(* CODESYS project CtaAppVerdichter_2.0.0.0.library
   Description: Verdichter Library der CTA
   Version: 2.0.0.0
   Title: CtaAppVerdichter
   Author: SIS
   DocFormat: reStructuredText
   Placeholder: CtaAppVerdichter
   LanguageModelAttribute: qualified-access-only
   CompiledLibraryCompatibilityVersion: CODESYS V3.5 SP16 Patch 3
   Company: CTA
   DefaultNamespace: CtaAppVerdichter

Project tree, tasks and I/O mapping:
  libraries: Standard, 3.5.18.0 (System); CtaAppBasic, 1.0.0.0 (CTA); CtaAppBmk, 2.0.0.0 (CTA); CtaAppReport, 2.0.0.0 (CTA); CtaSysConfig, 2.0.0.0 (CTA); CtaVisSymbols, 2.0.0.0 (CTA); CtaAppFilter, 1.0.0.0 (CTA); CtaAppHysterese, 1.0.0.0 (CTA); CtaSysMotor, 1.0.0.0 (CTA); CtaSysFU, 2.0.0.0 (CTA); VisuElemBase, 4.7.0.0 (System); CtaVisHelp, 2.0.0.0 (CTA); CtaAppDumper, 2.0.0.0 (CTA); CtaSysTypes, 1.0.0.0 (CTA); VisuDialogs, * (System); CtaAppEinsatzDiagramm, 2.0.0.0 (CTA); VisuSymbols, 4.5.0.0 (System); CtaSysLeistungventile, 2.0.0.0 (CTA); CtaAppInfluxLog, 1.0.0.1 (CTA); CtaSysIO, 2.0.0.0 (CTA); CtaAppModbusSpezifikation, 1.0.0.1 (CTA)
  40 Visualizations/
    ICON/
      VERDICHTER_RIGHT/
        VERDICHTER_RIGHT_BELOW/
          visualisation VIS_VERDICHTER_RIGHT_BELOW
          visualisation VIS_VERDICHTER_RigthBelowCheckIsEnabled
          visualisation VIS_VERDICHTER_RigthBelowCheckQuerry
        VERDICHTER_RIGHT_ABOVE/
          visualisation VIS_VERDICHTER_RigthAboveCheckQuerry
          visualisation VIS_VERDICHTER_RIGHT_ABOVE
          visualisation VIS_VERDICHTER_RigthAboveCheckIsEnabled
      VERDICHTER_BASE/
        visualisation CommandOn
        VALUE/
          visualisation ValueUpDwn
          visualisation ValueDwnUp
        ICON/
          visualisation Icon_Left
          visualisation Icon_Right
      VERDICHTER_LEFT/
        VERDICHTER_LEFT_BELOW/
          visualisation VIS_VERDICHTER_LEFT_BELOW
          visualisation VIS_VERDICHTER_LeftBelowCheckIsEnabled
          visualisation VIS_VERDICHTER_LeftBelowCheckQuerry
        VERDICHTER_LEFT_ABOVE/
          visualisation VIS_VERDICHTER_LEFT_ABOVE
          visualisation VIS_VERDICHTER_LeftAboveCheckIsEnabled
          visualisation VIS_VERDICHTER_LeftAboveCheckQuerry
    POPUP/
      visualisation POPUP_VERDICHTER
      PARAMETER/
        visualisation VIS_VERDICHTER_PARAMETER
        visualisation VIS_VERDICHTER_PARAMETER_LISTE
        VERDICHTER_ParameterBase/
          visualisation VIS_VERDICHTER_PARAMETER_BASE0
          visualisation VIS_VERDICHTER_PARAMETER_BASE
        VERDICHTER_Data/
          visualisation VIS_VERDICHTER_PARAMETER_DATA0
          visualisation VIS_VERDICHTER_PARAMETER_DATA
        VERDICHTER_Fuse/
          visualisation VIS_VERDICHTER_PARAMETER_FUSES0
          visualisation VIS_VERDICHTER_PARAMETER_FUSES
        VERDICHTER_IO/
          visualisation VIS_VERDICHTER_PARAMETER_IO0
          visualisation VIS_VERDICHTER_PARAMETER_IO1
          visualisation VIS_VERDICHTER_PARAMETER_IO
          visualisation VIS_VERDICHTER_PARAMETER_IO2
          visualisation VIS_VERDICHTER_PARAMETER_IO3
          visualisation VIS_VERDICHTER_PARAMETER_IO4
        VERDICHTER_InfluxDb/
          visualisation VIS_VERDICHTER_PARAMETER_TRENDLOG
          visualisation VIS_VERDICHTER_PARAMETER_TRENDLOG0
        visualisation VIS_ANTRIEB_POPUP_IO_ITF
      visualisation VIS_VERDICHTER_LISTE
      MANUAL/
        visualisation VIS_VERDICHTER_MANUAL
      OVERVIEW/
        visualisation VIS_VERDICHTER_OVERVIEW
        visualisation ResetVerdiTime
      BUS/
        visualisation VERDICHTER_BUS
        visualisation VERDICHTER_BUS_SW0_Detail
        visualisation VERDICHTER_BUS_CS
        visualisation VERDICHTER_BUS_SW1_Detail
        visualisation VERDICHTER_BUS_SW2_Detail
        visualisation VERDICHTER_BUS_SW3_Detail
      REPORTS/
        visualisation VIS_VERDICHTER_REPORTS
      IO/
        visualisation VIS_VERDICHTER_IO0
        visualisation VIS_VERDICHTER_IO
        visualisation VIS_VERDICHTER_IO1
  30 Program Organization Units/
    function block fbVerdichter [ST]: actConfig, proConfigError, proAtIconNr, P_scBase_fbtDelayOffToOn, P_scBase_fbtDelayOnToOn, P_scBase_fbrYMax, P_scBase_fbrYMin, P_scBase_fbxEnableFU, P_scBase_fbxEnable, P_scBase_fbxRegulatet, P_scData_fbudiOperatingHours, P_scData_fbudiOperationStarts, P_scFuse_fbxDoesAlarm, P_scFuse_fbxEnable, P_scFuse_fbxInputMb, P_scInfluxDb_fbxEnable, P_scIO_IsHand_fbxEnable, P_scIO_IsHand_fbxInputMb, P_scIO_IsNoError_fbxEnable, P_scIO_IsNoError_fbxInputMb, P_scIO_IsNoError_fbxDoesAlarm, P_scIO_IsNoError_fbtDelayStartSps, P_scIO_IsNoError_fbtDelayRun, P_scIO_IsNoError_fbiTypeOfAck, P_scIO_IsNoError_fbiMaxErrorRetryAllowed, P_scIO_IsOn_fbxInputMb, P_scIO_IsOn_fbxEnable, P_scIO_IsOn_fbtDelayStart, P_scIO_IsOn_fbxDoesAlarm, P_scIO_IsOn_fbtDelayRun, P_scIO_IsOn_fbiTypeOfAck, P_scIO_IsOn_fbiMaxErrorRetryAllowed, P_scIO_IsReady_fbxEnable, P_scIO_IsReady_fbxInputMb, P_scIO_IsValue_fbxInputMb, P_scIO_IsValue_fbxEnable, P_scIO_IsValue_fbxDoesAlarm, P_scIO_IsValue_fbtDelayStart, P_scIO_IsValue_fbtDelayRun, P_scIO_IsValue_fbiTypeOfAck, P_scIO_IsValue_fbiMaxErrorRetryAllowed, P_scIO_IsValue_fbrMaxDiff, P_scIO_RevisionSwitch_fbxEnable, P_scIO_RevisionSwitch_fbxInputMb, P_scManual_fbrManualOnY, P_scManual_fbuiManualState, P_scManual_fbxAlowManualOn, P_scVerdichterFuse_fbxDoesAlarm, P_scVerdichterFuse_fbxEnable, P_scVerdichterFuse_fbxInputMb, P_scFU_fbxReleaseMb, P_scFU_fbxSollWertMb, proRefToRonYDumper, actMbState, proModbusTest, proModbusStateWord, proIsError, proIsWarning, proIsRegulatet, proIsEnabled, actState, proMotorIsOn, proIsHandOnOrOff, proIsReady, proRestartLockAktive, proCommutingProtectionAktive, proRevisionSwitchOk, proCountedHours, proCountedStarts, proLeistung, proRestartLockTime, proCommutingProtectionTime, proIsOnY, proStateSymbol, proEnSymbol, proIsOn, proResetVerdiTime, proAuto, proHandOff, proHandOnY, proHardWareHandModulAktive, proHandOn, proGetDI_IsOn, metDI_IsOn, proNotShowDI_IsOn, proIsOn_ITF, metDI_RevisionSwitchOk, proNotShowDI_RevisionSwitchOk, proGetDI_RevisionSwitchOK, proRevisionSwitch_ITF, metDI_NoError, proNotShowDI_NoError, proGetDI_NoError, proNoError_ITF, proGetDI_FuseOK, metDI_ITF_FuseOK, proNotShowDI_FuseOk, proFuse_ITF, metDI_ITF_VerdichterHand, proNotShowDI_VerdichterHand, proGetDI_VerdichterHand, proHandModul_ITF, metDI_IsReady, proNotShowDI_Ready, proGetDI_IsReady, proReady_ITF, metDI_VerdichterFuseOk, proNotShowDI_VerdichterFuseOk, proGetDI_VerdichterFuseOk, proVerdichterFuse_ITF, metAI_ActualValue, proGetAI_ActualValue, proNotShowAI_ActualValue, proActualValue_ITF, proOnY_ITF, metAO_OnY, proDO_On, metDO_On, proOn_ITF, proOnY, proOn, actRestartAndCommutingLock, actPrioOfControll, actResetOnDisable, proOnHz, proEn, actTrendLog, actReport, proCountedError, proCountedInfo, proCountedWarning, proITF_REPORTMANAGER, proLockDown, proAvailable, proAcknowledge, proITF_EINSATZGRENZE, proITF_FU, actFU, proITF_LEISTUNGVENTILE, actLeistungsventile
    function fcGetBigerStringValue [ST]
    function fcCheckQuerryAndIconReturn [ST]
  00000000-0000-0000-0000-000000000000|D:\CoDeSys\LibrariesV3\trunk\Intern\CAA\CAA Template\3.4.0.0 draft\Placeholder.xml
  00000000-0000-0000-0000-000000000000|D:\CoDeSys\LibrariesV3\trunk\Intern\CAA\CAA Template\3.2.0.3 draft\Prefix.pdf
  00000000-0000-0000-0000-000000000000|D:\CoDeSys\LibrariesV3\trunk\Intern\CAA\CAA Template\3.5.2.0 draft\Placeholder.xml
  20 Structs/
    Verdichter/
      FU/
        data type scFU
      data type scParameter
      STATE/
        data type scInVerdichterHand
        data type scInVerichterActualValue
        data type scInVerdiRevisionSwitch
        data type scInVerdichterReady
        data type scInVerdichterNoError
        data type scInVerdichterOn
      BASE/
        data type scBase
      DATA/
        data type scData
      FUSE/
        data type scVerdichterFuse
        data type scFuse
      InfluxDb/
        data type scInfluxDb
      MANUAL/
        data type scManual
    Einsatzgrenze/
      data type scParameterEinsatzgrenze
      Paint/
        data type scLinePoint
        data type scDiagrammSizePaint
      Parameter/
        data type scSlopValue1
        data type scSlopValue2
        data type scSlopValue3
        data type scSlopValue4
        data type scSlopValue5
        data type scSlopValue6
        data type scDiagrammSize
        data type scErrorWarning
  50 Images/
  10 Documenation/
    global variables VersionHistory
    global variables readMe
  21 Interface/
    interface ITF_VERDICHTER: proModbusTest, proModbusStateWord, P_scFU_fbxReleaseMb, P_scFU_fbxSollWertMb, proConfigError, proAtIconNr, P_scBase_fbxEnable, P_scBase_fbxRegulatet, P_scBase_fbxEnableFU, P_scBase_fbrYMax, P_scBase_fbrYMin, P_scBase_fbtDelayOnToOn, P_scBase_fbtDelayOffToOn, P_scData_fbudiOperatingHours, P_scData_fbudiOperationStarts, P_scFuse_fbxDoesAlarm, P_scFuse_fbxEnable, P_scFuse_fbxInputMb, P_scInfluxDb_fbxEnable, P_scIO_RevisionSwitch_fbxEnable, P_scIO_RevisionSwitch_fbxInputMb, P_scIO_IsReady_fbxEnable, P_scIO_IsReady_fbxInputMb, P_scIO_IsHand_fbxEnable, P_scIO_IsHand_fbxInputMb, P_scIO_IsOn_fbxInputMb, P_scIO_IsOn_fbxEnable, P_scIO_IsOn_fbtDelayStart, P_scIO_IsOn_fbxDoesAlarm, P_scIO_IsOn_fbtDelayRun, P_scIO_IsOn_fbiTypeOfAck, P_scIO_IsOn_fbiMaxErrorRetryAllowed, P_scIO_IsNoError_fbxEnable, P_scIO_IsNoError_fbxInputMb, P_scIO_IsNoError_fbxDoesAlarm, P_scIO_IsNoError_fbtDelayStartSps, P_scIO_IsNoError_fbtDelayRun, P_scIO_IsNoError_fbiTypeOfAck, P_scIO_IsNoError_fbiMaxErrorRetryAllowed, P_scIO_IsValue_fbxInputMb, P_scIO_IsValue_fbxEnable, P_scIO_IsValue_fbxDoesAlarm, P_scIO_IsValue_fbtDelayStart, P_scIO_IsValue_fbtDelayRun, P_scIO_IsValue_fbiTypeOfAck, P_scIO_IsValue_fbiMaxErrorRetryAllowed, P_scIO_IsValue_fbrMaxDiff, P_scManual_fbrManualOnY, P_scManual_fbuiManualState, P_scManual_fbxAlowManualOn, P_scVerdichterFuse_fbxDoesAlarm, P_scVerdichterFuse_fbxEnable, P_scVerdichterFuse_fbxInputMb, proRefToRonYDumper, proCountedError, proCountedInfo, proITF_REPORTMANAGER, proCountedWarning, proCountedHours, proCountedStarts, proGetDI_VerdichterHand, proNotShowDI_VerdichterHand, proHandModul_ITF, proGetAI_ActualValue, proNotShowAI_ActualValue, proActualValue_ITF, proNotShowDI_NoError, proGetDI_NoError, proNoError_ITF, proNotShowDI_RevisionSwitchOk, proGetDI_RevisionSwitchOK, proRevisionSwitch_ITF, proNotShowDI_IsOn, proGetDI_IsOn, proIsOn_ITF, proNotShowDI_VerdichterFuseOk, proGetDI_VerdichterFuseOk, proVerdichterFuse_ITF, proNotShowDI_FuseOk, proGetDI_FuseOK, proFuse_ITF, proNotShowDI_Ready, proGetDI_IsReady, proReady_ITF, proOn_ITF, proOnY_ITF, proLeistung, proIsOn, proIsOnY, proEnSymbol, proStateSymbol, proIsRegulatet, proIsHandOnOrOff, proRestartLockTime, proOn, proCommutingProtectionTime, proCommutingProtectionAktive, proRestartLockAktive, proIsReady, proAuto, proHandOn, proIsError, proIsWarning, proEn, proOnY, proHardWareHandModulAktive, proIsEnabled, proMotorIsOn, proHandOff, proRevisionSwitchOk, proHandOnY, proOnHz, proResetVerdiTime, proLockDown, proAvailable, proAcknowledge, proITF_EINSATZGRENZE, proITF_FU, proITF_LEISTUNGVENTILE
  11 Library Parameter/
    global variables Parameter
  12 Konstanten/
    global variables GlobalKonstant
  60 Textlisten/
    text list GlobalTextList
    text list Error
    text list Info
    text list Warnung
  13 Globale Variablen/
  5ce3da45-db07-42e7-a21c-a00fff4ed8f6|C:\Users\sis\Downloads\dip-switch.svg
  5ce3da45-db07-42e7-a21c-a00fff4ed8f6|C:\Users\sis\Downloads\lightning-bolt-circle.svg
  5ce3da45-db07-42e7-a21c-a00fff4ed8f6|C:\Users\sis\Downloads\sine-wave.svg
  5ce3da45-db07-42e7-a21c-a00fff4ed8f6|C:\Users\sis\Downloads\eye.svg
  5ce3da45-db07-42e7-a21c-a00fff4ed8f6|C:\Users\sis\Downloads\lan.svg
*)

// 20 Structs/Verdichter/scParameter
{attribute 'pack_mode' := '1'} 
TYPE scParameter :
    STRUCT
        scBase              		:   scBase;
        scFuse              		:   scFuse;
        scVerdichterFuse        	:   scVerdichterFuse;
        scInVerdiRevisionSwitch		:   scInVerdiRevisionSwitch;
        scInVerdichterReady     	:   scInVerdichterReady;
 		scInVerdichterHand      	:   scInVerdichterHand;   
        scInVerdichterOn    		:   scInVerdichterOn;
        scInVerdichterNoError   	:   scInVerdichterNoError;
        scInVerdichterActualValue  	:   scInVerichterActualValue;
        scManual            		:   scManual;
        scData              		:   scData;
        scInfluxDb          		:   scInfluxDb;       
		scFU						:	scFU;
    END_STRUCT
END_TYPE

// 20 Structs/Verdichter/STATE/scInVerdichterHand
{attribute 'pack_mode' := '1'} 
TYPE scInVerdichterHand :
    STRUCT
        fbxEnable                   : CtaSysConfig.fbBOOL;    
        fbxInputMb                  : CtaSysConfig.fbBOOL; 
    END_STRUCT
END_TYPE

// 20 Structs/Verdichter/STATE/scInVerichterActualValue
{attribute 'pack_mode' := '1'} 
TYPE scInVerichterActualValue :
    STRUCT
        fbxEnable                    : CtaSysConfig.fbBOOL;
        fbxInputMb                   : CtaSysConfig.fbBOOL;   
        fbxDoesAlarm                 : CtaSysConfig.fbBOOL;  
        fbrMaxDiff                   : CtaSysConfig.fbREAL;
        fbtDelayStart                : CtaSysConfig.fbTIME;
        fbtDelayRun                  : CtaSysConfig.fbTIME;
		fbiTypeOfAck				 : CtaSysConfig.fbINT;
		fbiMaxErrorRetryAllowed		 : CtaSysConfig.fbINT;          
    END_STRUCT
END_TYPE

// 20 Structs/Verdichter/STATE/scInVerdiRevisionSwitch
{attribute 'pack_mode' := '1'} 
TYPE scInVerdiRevisionSwitch :
    STRUCT
        fbxEnable                   : CtaSysConfig.fbBOOL;
        fbxInputMb                  : CtaSysConfig.fbBOOL;           
    END_STRUCT
END_TYPE

// 20 Structs/Verdichter/STATE/scInVerdichterReady
{attribute 'pack_mode' := '1'} 
TYPE scInVerdichterReady :
    STRUCT
        fbxEnable                    : CtaSysConfig.fbBOOL;
        fbxInputMb                   : CtaSysConfig.fbBOOL;
		fbxDoesAlarm				 : CtaSysConfig.fbBOOL;
		fbtDelayStart				 : CtaSysConfig.fbTIME;
		fbtDelayRun					 : CtaSysConfig.fbTIME;
		fbiTypeOfAck				 : CtaSysConfig.fbINT;
		fbiMaxErrorRetryAllowed		 : CtaSysConfig.fbINT;          
    END_STRUCT
END_TYPE

// 20 Structs/Verdichter/STATE/scInVerdichterNoError
{attribute 'pack_mode' := '1'} 
TYPE scInVerdichterNoError :
    STRUCT
        fbxEnable                    : CtaSysConfig.fbBOOL;
        fbxInputMb                   : CtaSysConfig.fbBOOL;   
        fbxDoesAlarm                 : CtaSysConfig.fbBOOL;  
        fbtDelayStartSps             : CtaSysConfig.fbTIME;
        fbtDelayRun                  : CtaSysConfig.fbTIME; 
        fbiTypeOfAck                 : CtaSysConfig.fbINT; 
        fbiMaxErrorRetryAllowed      : CtaSysConfig.fbINT; 
    END_STRUCT
END_TYPE

// 20 Structs/Verdichter/STATE/scInVerdichterOn
{attribute 'pack_mode' := '1'} 
TYPE scInVerdichterOn :
    STRUCT
        fbxEnable                    : CtaSysConfig.fbBOOL;
        fbxInputMb                   : CtaSysConfig.fbBOOL;   
        fbxDoesAlarm                 : CtaSysConfig.fbBOOL;  
        fbtDelayStart                : CtaSysConfig.fbTIME;
        fbtDelayRun                  : CtaSysConfig.fbTIME; 
        fbiTypeOfAck                 : CtaSysConfig.fbINT;   
        fbiMaxErrorRetryAllowed      : CtaSysConfig.fbINT;      
    END_STRUCT
END_TYPE

// 20 Structs/Verdichter/BASE/scBase
{attribute 'pack_mode' := '1'} 
TYPE scBase :
    STRUCT
        fbxEnable       :   CtaSysConfig.fbBOOL;
        fbxRegulatet    :   CtaSysConfig.fbBOOL;
        fbxEnableFU   	:   CtaSysConfig.fbBOOL;
        fbrYMin         :   CtaSysConfig.fbREAL;
        fbrYMax         :   CtaSysConfig.fbREAL;
        fbtDelayOffToOn :   CtaSysConfig.fbTIME;
        fbtDelayOnToOn 	:   CtaSysConfig.fbTIME;
    END_STRUCT
END_TYPE

// 20 Structs/Verdichter/DATA/scData
{attribute 'pack_mode' := '1'} 
TYPE scData :
    STRUCT
        fbudiOperationStarts    :   CtaSysConfig.fbUDINT;
        fbudiOperatingHours     :   CtaSysConfig.fbUDINT;       
    END_STRUCT
END_TYPE

// 20 Structs/Verdichter/FUSE/scVerdichterFuse
{attribute 'pack_mode' := '1'} 
TYPE scVerdichterFuse :
    STRUCT
        fbxEnable             : CtaSysConfig.fbBOOL;
        fbxInputMb            : CtaSysConfig.fbBOOL;
        fbxDoesAlarm          : CtaSysConfig.fbBOOL;      
    END_STRUCT
END_TYPE

// 20 Structs/Verdichter/FUSE/scFuse
{attribute 'pack_mode' := '1'} 
TYPE scFuse :
    STRUCT
        fbxEnable               : CtaSysConfig.fbBOOL;
        fbxInputMb              : CtaSysConfig.fbBOOL;
        fbxDoesAlarm            : CtaSysConfig.fbBOOL;
    END_STRUCT
END_TYPE

// 20 Structs/Verdichter/InfluxDb/scInfluxDb
{attribute 'pack_mode' := '1'} 
TYPE scInfluxDb :
    STRUCT
        fbxEnable       :   CtaSysConfig.fbBOOL;
    END_STRUCT
END_TYPE

// 20 Structs/Verdichter/MANUAL/scManual
{attribute 'pack_mode' := '1'} 
TYPE scManual :
    STRUCT
        fbxAlowManualOn         : CtaSysConfig.fbBOOL;    
        fbuiManualState         : CtaSysConfig.fbUINT;            // 0 = Auto ; 1 = Manual Off 2 = Manual On
        fbrManualOnY            : CtaSysConfig.fbREAL; 
    END_STRUCT
END_TYPE

// 20 Structs/Verdichter/FU/scFU
TYPE scFU :
	STRUCT
		fbxReleaseMb            : CtaSysConfig.fbBOOL;
		fbxSollWertMb           : CtaSysConfig.fbBOOL;
	END_STRUCT
END_TYPE

// 20 Structs/Einsatzgrenze/scParameterEinsatzgrenze
TYPE scParameterEinsatzgrenze :
    STRUCT
        scDiagrammSize              :   scDiagrammSize;
        fbrMinTc					:	CtaSysConfig.fbREAL;							        // Minimale Kondensationstemperatur [°C] 
        fbrMaxTc					:	CtaSysConfig.fbREAL;							        // Maximale Kondensationstemperatur [°C] 
        fbrMinTo					:	CtaSysConfig.fbREAL;							        // Minimale Verdampfungstemperatur  [°C]
        fbrMaxTo					:	CtaSysConfig.fbREAL; 							        // Maximale Verdampfungstemperatur  [°C]             
        scSlopValue1                :   scSlopValue1;         
        scSlopValue2                :   scSlopValue2;
        scSlopValue3                :   scSlopValue3;
        scSlopValue4                :   scSlopValue4;
        scSlopValue5                :   scSlopValue5;
        scSlopValue6                :   scSlopValue6;        
        scErrorWarning              :   scErrorWarning; 
    END_STRUCT
END_TYPE

// 20 Structs/Einsatzgrenze/Paint/scLinePoint
TYPE scLinePoint :
    STRUCT
        rP1X        :   REAL;
        rP1Y        :   REAL;      
    END_STRUCT
END_TYPE

// 20 Structs/Einsatzgrenze/Paint/scDiagrammSizePaint
TYPE scDiagrammSizePaint :
    STRUCT
        rYMax   :   REAL;
        rYMin   :   REAL;
        rXMax   :   REAL;
        rXMin   :   REAL;    
    END_STRUCT
END_TYPE

// 20 Structs/Einsatzgrenze/Parameter/scSlopValue1
TYPE scSlopValue1 :
    STRUCT
        fbrTcL			    :	CtaSysConfig.fbREAL;							        // Punkt  1 Kompressor-Auslegungsdiagramm [°C] 
        fbrT0L              :   CtaSysConfig.fbREAL;	                                // Punkt  2 Kompressor-Auslegungsdiagramm [°C]
        fbrT0R  		    :	CtaSysConfig.fbREAL;							        // Punkt  3 Kompressor-Auslegungsdiagramm [°C]        
    END_STRUCT
END_TYPE

// 20 Structs/Einsatzgrenze/Parameter/scSlopValue2
TYPE scSlopValue2 :
    STRUCT
        fbrTcR			    :	CtaSysConfig.fbREAL;							        // Punkt  4 Kompressor-Auslegungsdiagramm [°C] 
        fbrT0R  		    :	CtaSysConfig.fbREAL;							        // Punkt  5 Kompressor-Auslegungsdiagramm [°C]        
    END_STRUCT
END_TYPE

// 20 Structs/Einsatzgrenze/Parameter/scSlopValue3
TYPE scSlopValue3 :
    STRUCT
        fbrTcU			    :	CtaSysConfig.fbREAL;							        // Punkt  6 Kompressor-Auslegungsdiagramm [°C] 
    END_STRUCT
END_TYPE

// 20 Structs/Einsatzgrenze/Parameter/scSlopValue4
TYPE scSlopValue4 :
    STRUCT
        fbrTcL			    :	CtaSysConfig.fbREAL;							        // Punkt  7 Kompressor-Auslegungsdiagramm [°C]         
    END_STRUCT
END_TYPE

// 20 Structs/Einsatzgrenze/Parameter/scSlopValue5
TYPE scSlopValue5 :
    STRUCT
        fbrT0L			    :	CtaSysConfig.fbREAL;							        // Punkt  8 Kompressor-Auslegungsdiagramm [°C] 
        fbrT0R  			:	CtaSysConfig.fbREAL;							        // Punkt  9 Kompressor-Auslegungsdiagramm [°C]                
    END_STRUCT
END_TYPE

// 20 Structs/Einsatzgrenze/Parameter/scSlopValue6
TYPE scSlopValue6 :
    STRUCT
        fbrTcO			    :	CtaSysConfig.fbREAL;							        // Punkt 10 Kompressor-Auslegungsdiagramm [°C]                 
    END_STRUCT
END_TYPE

// 20 Structs/Einsatzgrenze/Parameter/scDiagrammSize
TYPE scDiagrammSize :
    STRUCT
        fbrYMax   :   CtaSysConfig.fbREAL;
        fbrYMin   :   CtaSysConfig.fbREAL;
        fbrXMax   :   CtaSysConfig.fbREAL;
        fbrXMin   :   CtaSysConfig.fbREAL;    
    END_STRUCT
END_TYPE

// 20 Structs/Einsatzgrenze/Parameter/scErrorWarning
TYPE scErrorWarning :
    STRUCT
        fbxEnEW1          :   CtaSysConfig.fbBOOL;
        fbxEnEW2          :   CtaSysConfig.fbBOOL;
        fbxEnEW3          :   CtaSysConfig.fbBOOL;
        fbxEnEW4          :   CtaSysConfig.fbBOOL;
        fbxEnEW5          :   CtaSysConfig.fbBOOL;
        fbxEnEW6          :   CtaSysConfig.fbBOOL;
        fbxEnEW7          :   CtaSysConfig.fbBOOL;
        fbtDelayWarning   :   CtaSysConfig.fbTIME;
        fbiAnzError       :   CtaSysConfig.fbINT;
        fbtDelayError     :   CtaSysConfig.fbTIME;
        fbtCountReset     :   CtaSysConfig.fbTIME;
    END_STRUCT
END_TYPE

// 10 Documenation/VersionHistory
(* 

.. image:: ../../Images/CTA_Logo.jpg
   :align: right
   :width: 15% 

**Vorlage**   


============ =========== =========== ============================================
**Date**     **Version** **Author**  **Change**
------------ ----------- ----------- --------------------------------------------
04.03.2021   0.0.0.0     SIS         Vorlage erstellt

============ =========== =========== ============================================


*)
VAR_GLOBAL
    stInfo : STRING:= '0.0.0.0, Vorlage, CTA';
END_VAR

// 10 Documenation/readMe
(*

**ReadMe**
 
|	**Empfehlung**
|
|	Bibliothek CtaAppVerdichter zur Ansteuerung von Verdichtern
|	Instanzieren Sie den CtaAppVerdichter.fbVerdichter in ihrem Funktionsbaustein oder POU beispielsweise als fbVerdiX. (X = Nr.)
|	Instanzieren Sie den CtaAppVerdichter.fbEinsatzgrenze in ihrem Funktionsbaustein oder POU beispielsweise als fbVerdiXEinsatzGr. (X = Nr des Verdicheters)
|	Deklarieren Sie die Struktur Variable welche als Parameter und zur ansteuerung dienen wie im Code beispiel.
|  
| *Beispiel* 

+-----------------------+---------------------------------------------------------------------------------------------------------------------------------------------------------------------------------------------------------------------------------------------------------------------------------------------------------------------------------------------------------------------------------------------------------------------------------------+
| Beschreibung          |  Code                                                                                                                                                                                                                                                                                                                                                                                                                                 |
+=======================+=======================================================================================================================================================================================================================================================================================================================================================================================================================================+
| Pou oder SmFb         | .. code-block:: codesys                                                                                                                                                                                                                                                                                                                                                                                                               |
|                       |                                                                                                                                                                                                                                                                                                                                                                                                                                       |
|                       |	// Deklaration als VAR im POU oder dem selbsterstellten Funktionsbaustein                                                                                                                                                                                                                                                                                                                                                       	|
|                       |   VAR   																																																																																																								|
|						|	    (*Verdichter1*)																																																		 																																																			|
|						|		fbVerdi1			: CtaAppVerdichter.fbVerdichter;                                                                                                                                                                                                                                                                                                                                                              				|
|						|	    (*Einsatzgrenze Verdichter1*)																																																		 																																															|
|						|		fbVerdi1EinsatzGr	: CtaAppVerdichter.fbEinsatzgrenze;                                                                                                                                                                                                                                                                                                                                                              			|
| 						|	END_VAR                                                                                                                                                                                                                                                                                                                                                                                                                         	|
+-----------------------+---------------------------------------------------------------------------------------------------------------------------------------------------------------------------------------------------------------------------------------------------------------------------------------------------------------------------------------------------------------------------------------------------------------------------------------+
| Code für Init         | .. code-block:: codesys                                                                                                                                                                                                                                                                                                                                                                                                               |
|                       |   																																																																																																									|
| 						|	// Kopieren des nachfolgenden Codes in eine Action zur Initialisierung der Parameter. Zum Beispiel actConfig.																																																																														|
|                       |	{region "Parameter Verdichter1"}                                                                                                                                                                                                                                                                                                                                                                                                    |
| 						|		(*Basis*)																																																																																																						|
|						|		fbVerdi1.scParameter.scBase.fbxEnable               					(_wertInit :=  TRUE																			);		//P1 Ein- Ausschalten des Verdichters																																																				|
|						|		fbVerdi1.scParameter.scBase.fbxRegulatet								(_wertInit :=  TRUE																			);		//P2 Verdichter ist geregelt / nicht geregelt																																																		|
|						|		fbVerdi1.scParameter.scBase.fbxEnableFU									(_wertInit :=  TRUE																			);		//P3 Ansteuerung oder Signalauswertung über Modbus																																																	|
|						|		fbVerdi1.scParameter.scBase.fbrYMin										(_wertInit :=   0.0									, _minInit :=   0.0, _maxInit := 100.0	);		//P4 Minimaler Stellwert des Verdichters																																																			|
|						|		fbVerdi1.scParameter.scBase.fbrYMax										(_wertInit := 100.0									, _minInit :=   0.0, _maxInit := 100.0	);		//P5 Maximaler Stellwert des Verdichters																																																			|
|						|		fbVerdi1.scParameter.scBase.fbtDelayOffToOn								(_wertInit := T#30S									, _minInit :=      , _maxInit :=		);		//P6 Sperrzeit des Verdichters																																																						|
|						|		fbVerdi1.scParameter.scBase.fbtDelayOnToOn								(_wertInit := T#60S									, _minInit :=	   , _maxinit :=		);		//P7 Pendelschutz des Verdichters																																																					|
|						|		(*Sicherungen*)																																																		 																																																			|
|						|		fbVerdi1.scParameter.scFuse.fbxEnable									(_wertInit := FALSE																			);		//P8 Sicherung ist vorhanden / nicht vorhanden																	    																																|
|						|		fbVerdi1.scParameter.scFuse.fbxInputMb									(_wertInit := FALSE																			);		//P9 Ansteuerung oder Signalauswertung über Modbus																												    																				|
|						|		fbVerdi1.scParameter.scFuse.fbxDoesAlarm								(_wertInit := FALSE																			);		//P10 Abfallendes Signal löst Fehler aus																											    																							|
|						|		(*Motorsicherung*)																																																											 																																	  								|
|						|		fbVerdi1.scParameter.scVerdichterFuse.fbxEnable							(_wertInit := FALSE																			);		//P11 Leistungsschutzschalter ist vorhanden / nicht vorhanden																    																													|
|						|		fbVerdi1.scParameter.scVerdichterFuse.fbxInputMb						(_wertInit := FALSE																			);		//P12 Ansteuerung oder Signalauswertung über Modbus																																								   	 								|
|						|		fbVerdi1.scParameter.scVerdichterFuse.fbxDoesAlarm						(_wertInit := FALSE																			);		//P13 Abfallendes Signal löst Fehler aus																														    																				|
|						|		(*Revisionsschalter*)																																																											 																																							    |
|						|		fbVerdi1.scParameter.scInVerdiRevisionSwitch.fbxEnable					(_wertInit := FALSE																			);		//P14 Revisionsschalter ist vorhanden / nicht vorhanden																																				    											|
|						|		fbVerdi1.scParameter.scInVerdiRevisionSwitch.fbxInputMb					(_wertInit := FALSE																			);		//P15 Ansteuerung oder Signalauswertung über Modbus																																		    														|
|						|		(*Handmodul*)																																																		 																																																		    |
|						|		fbVerdi1.scParameter.scInVerdichterHand.fbxEnable						(_wertInit := FALSE																			);		//P40 Handmodul ist vorhanden / nicht vorhanden																																																		|
|						|		fbVerdi1.scParameter.scInVerdichterHand.fbxInputMb						(_wertInit := FALSE																			);		//P41 Ansteuerung oder Signalauswertung über Modbus																																																	|
|						|		(*Ready- Input*)																																																																																																		    	|
|						|		fbVerdi1.scParameter.scInVerdichterReady.fbxEnable						(_wertInit := FALSE																			);		//P16 Readysignal ist vorhanden / nicht vorhanden																																	    															|
|						|		fbVerdi1.scParameter.scInVerdichterReady.fbxInputMb						(_wertInit := FALSE																			);		//P17 Ansteuerung oder Signalauswertung über Modbus																																										    						|
|						|		(*Betriebsrückmeldung*)																																																										 																																								    |
|						|		fbVerdi1.scParameter.scInVerdichterOn.fbxEnable							(_wertInit := FALSE																			);		//P18 Betriebsrückmeldung ist vorhanden / nicht vorhanden																														   																	|
|						|		fbVerdi1.scParameter.scInVerdichterOn.fbxInputMb						(_wertInit := FALSE																			);		//P19 Ansteuerung oder Signalauswertung über Modbus																																								    								|
|						|		fbVerdi1.scParameter.scInVerdichterOn.fbxDoesAlarm						(_wertInit := FALSE																			);		//P20 Fehlendes oder abfallendes Signal löst Fehler aus				   																																												|
|						|		fbVerdi1.scParameter.scInVerdichterOn.fbtDelayStart						(_wertInit := T#00S									, _minInit :=      , _maxInit :=  		);		//P21 Verzögerung der Fehlerausgabe nach Start																						   																												|
|						|		fbVerdi1.scParameter.scInVerdichterOn.fbtDelayRun						(_wertInit := T#00S									, _minInit :=      , _maxInit :=  		);		//P22 Verzögerung der Fehlerausgabe während Betrieb															    																																	|
|						|		fbVerdi1.scParameter.scInVerdichterOn.fbiTypeOfAck						(_wertInit :=     1 								, _minInit :=     0, _maxInit :=    2	);		//P23 Art der Quittierung des Fehlers (auto, quittierend, quittierend bid n Meldung																																									|
|						|		fbVerdi1.scParameter.scInVerdichterOn.fbiMaxErrorRetryAllowed			(_wertInit :=     3									, _minInit :=     0, _maxInit :=    5	);		//P24 Maximale Anzahl Wiederholungen bis zur Sperrung der Anlage																																													|
|						|		(*Fehler- Input*)																																																																																																			    |
|						|		fbVerdi1.scParameter.scInVerdichterNoError.fbxEnable					(_wertInit := FALSE																			);		//P25 Fehlerinput ist vorhanden / nicht vorhanden																																		    														|
|						|		fbVerdi1.scParameter.scInVerdichterNoError.fbxInputMb					(_wertInit := FALSE																			);		//P26 Ansteuerung oder Signalauswertung über Modbus																																																	|
|						|		fbVerdi1.scParameter.scInVerdichterNoError.fbxDoesAlarm					(_wertInit := FALSE																			);		//P27 Fehlendes oder abfallendes Signal löst Fehler aus				   																																												|
|						|		fbVerdi1.scParameter.scInVerdichterNoError.fbtDelayStartSps				(_wertInit :=  T#0S									, _minInit :=      , _maxInit :=  		);		//P28 Verzögerung der Fehlerausgabe nach Start																																																		|
|						|		fbVerdi1.scParameter.scInVerdichterNoError.fbtDelayRun					(_wertInit :=  T#0S									, _minInit :=      , _maxInit :=  		);		//P29 Verzögerung der Fehlerausgabe während Betrieb																																																	|
|						|		fbVerdi1.scParameter.scInVerdichterNoError.fbiTypeOfAck					(_wertInit :=     1 								, _minInit :=     0, _maxInit :=    2	);		//P30 Art der Quittierung des Fehlers (auto, quittierend, quittierend bid n Meldung																																									|
|						|		fbVerdi1.scParameter.scInVerdichterNoError.fbiMaxErrorRetryAllowed		(_wertInit :=     3 								, _minInit :=     0, _maxInit :=    5	);		//P31 Maximale Anzahl Wiederholungen bis zur Sperrung der Anlage																																										    		|
|						|		(*Ist - Wert*)																																																																																																				    |
|						|		fbVerdi1.scParameter.scInVerdichterActualValue.fbxEnable				(_wertInit := FALSE																			);		//P32 Rückmeldung des Istwerts ist vorhanden / nicht vorhanden																																														|
|						|		fbVerdi1.scParameter.scInVerdichterActualValue.fbxInputMb				(_wertInit := FALSE																			);		//P33 Ansteuerung oder Signalauswertung über Modbus																																																	|
|						|		fbVerdi1.scParameter.scInVerdichterActualValue.fbxDoesAlarm				(_wertInit := FALSE																			);		//P34 Unter oder überschreitung der Maximal erlaubten Differenz löst Fehler aus				   																																						|
|						|		fbVerdi1.scParameter.scInVerdichterActualValue.fbrMaxDiff				(_wertInit :=   0.0									, _minInit :=		, _maxInit :=		);		//P34 Maximal erlaubte Differenz des Stell- zum Istwert  			   																																												|
|						|		fbVerdi1.scParameter.scInVerdichterActualValue.fbtDelayStart			(_wertInit := T#00S									, _minInit :=      , _maxInit :=    	);		//P36 Verzögerung der Fehlerausgabe nach Start																																																		|
|						|		fbVerdi1.scParameter.scInVerdichterActualValue.fbtDelayRun				(_wertInit := T#00S									, _minInit :=      , _maxInit :=    	);		//P37 Verzögerung der Fehlerausgabe während Betrieb																																																	|
|						|		fbVerdi1.scParameter.scInVerdichterActualValue.fbiTypeOfAck				(_wertInit :=     1 								, _minInit :=     0, _maxInit :=    2	);		//P38 Art der Quittierung des Fehlers (auto, quittierend, quittierend bid n Meldung																																									|
|						|		fbVerdi1.scParameter.scInVerdichterActualValue.fbiMaxErrorRetryAllowed 	(_wertInit :=     3									, _minInit :=     0, _maxInit :=    5	);		//P39 Maximale Anzahl Wiederholungen bis zur Sperrung der Anlage																																													|
|						|		(*Manuelle Ansteuerung*)																																																																																																	    |
|						|		fbVerdi1.scParameter.scManual.fbxAlowManualOn							(_wertInit :=  TRUE																			);		//P42 Handansteuerung zulassen / nicht zulassen																																																		|
|						|		fbVerdi1.scParameter.scManual.fbuiManualState							(_wertInit := 	  0									, _minInit :=     0, _maxInit :=    2	);		//P43 Ansteuerungsmodus des Ventils (auto, manuell, gesperrt)																																														|
|						|		fbVerdi1.scParameter.scManual.fbrManualOnY								(_wertInit := 	  0									, _minInit :=     0, _maxInit :=  100	);		//P44 Manueller Stellwert für den Antrieb																																																			|
|						|		(*Betriebsdaten*)																																																																																																			    |
|						|		fbVerdi1.scParameter.scData.fbudiOperationStarts						(_wertInit := 	  0									, _minInit :=     0, _maxInit :=    0	);		//P45 Betriebsstarts des Verdichters																																																				|
|						|		fbVerdi1.scParameter.scData.fbudiOperatingHours							(_wertInit :=     0									, _minInit :=     0, _maxInit :=    0	);		//P46 Betriebsstunden des Verdichters																																																				|
|						|		(*Trendlog*)																																																																																																					|
|						|		fbVerdi1.scParameter.scInfluxDb.fbxEnable								(_wertInit :=  TRUE																			);		//P47 Aktiverung / Deaktivierung der Trenddaten 																																																	|
|						|		(* FU *)																																																																																																						|
|						|		fbVerdi1.scParameter.scFU.fbxReleaseMb									(_wertInit := FALSE																			);		//P48 TRUE = Freigabe über Modbus																																																					|
|						|		fbVerdi1.scParameter.scFU.fbxSollWertMb									(_wertInit := FALSE																			);		//P49 TRUE = Sollwert über Modbus																																																					|
|						|	{endregion}                                             	                                                                                                         																																																																|
|                       |	{region "Parameter Einsatzgrenzen Verdichter1"}                                                                                                                                                                                                                                                                                                                                                                                     |
| 						|		(*Diagrammgrösse*)																																																																																																				|
|						|		fbVerdi1EinsatzGr.scParaData.scDiagrammSize.fbrYMax               		(_wertInit :=   0.0									, _minInit :=		, _maxInit :=		);		//P1 Diagrammgrösse Y Achse Max																																																						|
|						|		fbVerdi1EinsatzGr.scParaData.scDiagrammSize.fbrYMin						(_wertInit :=   0.0									, _minInit :=		, _maxInit :=		);		//P2 Diagrammgrösse Y Achse Min																																																						|
|						|		fbVerdi1EinsatzGr.scParaData.scDiagrammSize.fbrXMax						(_wertInit :=   0.0									, _minInit :=		, _maxInit :=		);		//P3 Diagrammgrösse X Achse Max																																																						|
|						|		fbVerdi1EinsatzGr.scParaData.scDiagrammSize.fbrXMin						(_wertInit :=   0.0									, _minInit :=		, _maxInit :=		);		//P4 Diagrammgrösse X Achse Min																																																						|
|						|		(*Min Max Tc & To*)																																																		 																																																		|
|						|		fbVerdi1EinsatzGr.scParaData.fbrMinTc									(_wertInit :=   0.0									, _minInit :=		, _maxInit :=		);		//P5 Max Tc																																																											|
|						|		fbVerdi1EinsatzGr.scParaData.fbrMaxTc									(_wertInit :=   0.0									, _minInit :=		, _maxInit :=		);		//P6 Min Tc																																																											|
|						|		fbVerdi1EinsatzGr.scParaData.fbrMinTo									(_wertInit :=   0.0									, _minInit :=		, _maxInit :=		);		//P7 Max To																																																											|
|						|		fbVerdi1EinsatzGr.scParaData.fbrMaxTo									(_wertInit :=   0.0									, _minInit :=		, _maxInit :=		);		//P8 Min To																																																											|
|						|		(*Slop Value 1*)																																																		 																																																		|
|						|		fbVerdi1EinsatzGr.scParaData.scSlopValue1.fbrTcL						(_wertInit :=   0.0									, _minInit :=		, _maxInit :=		);		//P9 Slop Value 1 Tc Links																	    																																					|
|						|		fbVerdi1EinsatzGr.scParaData.scSlopValue1.fbrT0L						(_wertInit :=   0.0									, _minInit :=		, _maxInit :=		);		//P10 Slop Value 1 To Links																												    																										|
|						|		fbVerdi1EinsatzGr.scParaData.scSlopValue1.fbrT0R						(_wertInit :=   0.0									, _minInit :=		, _maxInit :=		);		//P11 Slop Value 1 To Rechts																											    																										|
|						|		(*Slop Value 2*)																																																										 																																	  									|
|						|		fbVerdi1EinsatzGr.scParaData.scSlopValue2.fbrTcR						(_wertInit :=   0.0									, _minInit :=		, _maxInit :=		);		//P12 Slop Value 2 Tc Rechts																    																																					|
|						|		fbVerdi1EinsatzGr.scParaData.scSlopValue2.fbrT0R						(_wertInit :=   0.0									, _minInit :=		, _maxInit :=		);		//P13 Slop Value 2 To Rechts																																								   	 													|
|						|		(*Slop Value 3*)																																																											 																																							    	|
|						|		fbVerdi1EinsatzGr.scParaData.scSlopValue3.fbrTcU						(_wertInit :=   0.0									, _minInit :=		, _maxInit :=		);		//P14 Slop Value 3 Tc Unten																														    																								|
|						|		(*Slop Value 4*)																																																											 																																							    	|
|						|		fbVerdi1EinsatzGr.scParaData.scSlopValue4.fbrTcL						(_wertInit :=   0.0									, _minInit :=		, _maxInit :=		);		//P15 Slop Value 4 Tc Links																																				    																		|
|						|		(*Slop Value 5*)																																																		 																																																		|
|						|		fbVerdi1EinsatzGr.scParaData.scSlopValue5.fbrT0L						(_wertInit :=   0.0									, _minInit :=		, _maxInit :=		);		//P16 Slop Value 5 To Links																																		    																				|
|						|		fbVerdi1EinsatzGr.scParaData.scSlopValue5.fbrT0R						(_wertInit :=   0.0									, _minInit :=		, _maxInit :=		);		//P17 Slop Value 5 To Rechts																																		    																			|
|						|		(*Slop Value 6*)																																																		 																																																		|
|						|		fbVerdi1EinsatzGr.scParaData.scSlopValue6.fbrTcO						(_wertInit :=   0.0									, _minInit :=		, _maxInit :=		);		//P18 Slop Value 6 Tc Oben																																																							|
|						|		(*Error & Warnungen*)																																																																																																		    |
|						|		fbVerdi1EinsatzGr.scParaData.scErrorWarning.fbxEnEW1					(_wertInit := FALSE																			);		//P19 Überwachung Slop Value 1																																	    																				|
|						|		fbVerdi1EinsatzGr.scParaData.scErrorWarning.fbxEnEW2					(_wertInit := FALSE																			);		//P20 Überwachung Slop Value 2																																										    											|
|						|		fbVerdi1EinsatzGr.scParaData.scErrorWarning.fbxEnEW3					(_wertInit := FALSE																			);		//P21 Überwachung Slop Value 3																														   																								|
|						|		fbVerdi1EinsatzGr.scParaData.scErrorWarning.fbxEnEW4					(_wertInit := FALSE																			);		//P22 Überwachung Slop Value 4																																								    													|
|						|		fbVerdi1EinsatzGr.scParaData.scErrorWarning.fbxEnEW5					(_wertInit := FALSE																			);		//P23 Überwachung Slop Value 5				   																																																		|
|						|		fbVerdi1EinsatzGr.scParaData.scErrorWarning.fbxEnEW6					(_wertInit := FALSE																			);		//P24 Überwachung Slop Value 6																						   																																|
|						|		fbVerdi1EinsatzGr.scParaData.scErrorWarning.fbxEnEW7					(_wertInit := FALSE																			);		//P25 Überwachung Slop Value 7														    																																							|
|						|		fbVerdi1EinsatzGr.scParaData.scErrorWarning.fbtDelayWarning				(_wertInit := T#00S									, _minInit :=		, _maxInit :=		);		//P26 Warnungsverzögerung																																																							|
|						|		fbVerdi1EinsatzGr.scParaData.scErrorWarning.fbiAnzError					(_wertInit :=     0									, _minInit :=		, _maxInit :=		);		//P27 Anzahl Error Autoquittierungen																																																				|
|						|		fbVerdi1EinsatzGr.scParaData.scErrorWarning.fbtDelayError				(_wertInit := T#00S									, _minInit :=	    , _maxInit :=		);		//P28 Errorverzögerung																																																								|
|						|		fbVerdi1EinsatzGr.scParaData.scErrorWarning.fbtCountReset				(_wertInit := T#00S									, _minInit :=		, _maxInit :=		);		//P29 Reset des Zähler nach t																																																						|
|						|	{endregion}                                             	                                                                                                         																																																																|
+-----------------------+---------------------------------------------------------------------------------------------------------------------------------------------------------------------------------------------------------------------------------------------------------------------------------------------------------------------------------------------------------------------------------------------------------------------------------------+
*)                                                                                                                                                                                                                                                                                                                                                                                                                                                               
 VAR_GLOBAL                                                                                                                                                                                                                                                                                                                                                                                                                                                      
    xReadMeDone              :   BOOL;                                                                                                                                                                                                                                                                                                                                                                                                                           
END_VAR

// 11 Library Parameter/Parameter
{attribute 'qualified_only'}
VAR_GLOBAL CONSTANT
    iMaxVerdichter :   INT   := 60;         // Maximale Anzahl verwendeter AT-Bausteine    
END_VAR

// 12 Konstanten/GlobalKonstant
{attribute 'qualified_only'}
VAR_GLOBAL CONSTANT 	
	stReportTextListError   : CtaAppReport.stReportTextList := 'CtaAppVerdichter.Error';
	stReportTextListWarning : CtaAppReport.stReportTextList := 'CtaAppVerdichter.Warnung';
	stReportTextListInfo    : CtaAppReport.stReportTextList := 'CtaAppVerdichter.Info';	
    uiMaxParameter          : UINT := 47;
END_VAR

// 30 Program Organization Units/fbVerdichter
FUNCTION_BLOCK fbVerdichter EXTENDS CtaAppBmk.fbBMK IMPLEMENTS ITF_VERDICHTER 
VAR_INPUT
    xRelease                    :   BOOL;
    rRelease                    :   REAL;
	xReadyExt					:	BOOL;
    xSafetyStop                 :   BOOL;
	scHzParameter				:	CtaSysTypes.scHzParameter;
END_VAR
                     
VAR_OUTPUT                      
    (* Commmands *)               
    xOn                         :   BOOL; 
    rOnY                        :   REAL;	
    (* State Out*)              
    xIsOn                       :   BOOL;
	rOnHz						:	REAL;
	xIsReady					:	BOOL;	
END_VAR                 
VAR                     
    (* State Intern*)      
    scEWI                       :   CtaAppReport.scReportNr;                 
    xIsWarning                  :   BOOL;
    _xIsWarning                 :   BOOL;
    xIsError                    :   BOOL;
    _xIsError                   :   BOOL;
    xIsRegulatet                :   BOOL;
    xIsEnabled                  :   BOOL;
    xIsHand                     :   BOOL;
    xIsHandOn                   :   BOOL;
    xIsHandOff                  :   BOOL;
    xIsAuto                     :   BOOL;   
    xConfigError                :   BOOL;
	uiIconNr					:	UINT;	
	xOnOld						:	BOOL;
	rOnYVisu					:	REAL;
	fbDumperRonY				:	CtaAppDumper.fbDumper;	
	(* ITF OUT*)
	ITF_xOn						:	CtaSysIO.ITF_IO;
	ITF_rOnY					:	CtaSysIO.ITF_IO;	
    (* Inputs *)
	(*Fuse*)
    xFuseOk                     :   BOOL;
    xInFuseOk                   :   BOOL;
    xInFuseOkMb                 :   BOOL;
	ITF_Fuse					:	CtaSysIO.ITF_IO; 
 	(*Motorfuse*)
    xVerdichterFuseOk           :   BOOL;    
    xInVerdichterFuseOk         :   BOOL;
    xInVerdichterFuseOkMb       :   BOOL;
	ITF_VerdichterFuse			:	CtaSysIO.ITF_IO; 
	(*Motorerror*)
    xVerdichterNoError          :   BOOL;   
    xInVerdichterNoError        :   BOOL;
    xInVerdichterNoErrorMb      :   BOOL;
	ITF_VerdichterNoError		:	CtaSysIO.ITF_IO;
	(*MotorReady*)
    xVerdichterIsReady          :   BOOL;
    xInVerdichterIsReady        :   BOOL;
    xInVerdichterIsReadyMb      :   BOOL;
	ITF_VerdichterIsReady		:	CtaSysIO.ITF_IO;
	(*Motor status*)
    xVerdichterIsOn             :   BOOL;
    xInVerdichterIsOn           :   BOOL;
    xInVerdichterIsOnMb         :   BOOL;
	ITF_VerdichterIsOn			:	CtaSysIO.ITF_IO;
	(*Revisionsschalter*)
    xVerdiRevisionSwitchOff     :   BOOL;
    xVerdiRevisionSwitchOn      :   BOOL;
    xInVerdiRevisionSwitchOn    :   BOOL;   
    xInVerdiRevisionSwitchOnMb  :   BOOL;
	ITF_RevisionSwitch			:	CtaSysIO.ITF_IO;
	(*Handansteuerung*) 
    xVerdichterHand             :   BOOL;
    xInVerdichterHand           :   BOOL;
    xInVerdichterHandMb         :   BOOL;
	ITF_VerdichterHand		    :	CtaSysIO.ITF_IO;
	(*Aktueller Wert*)
	rActualValue				:	REAL;
    rInActualValue              :   REAL;
	rInActualValueModbus		:	REAL;
	ITF_ActualValue				:	CtaSysIO.ITF_IO; 
    (* Motor *)
    rVerdichterReleaseY        	:   REAL;
    xReleaseVerdichter          :   BOOL;
    rReleaseScaled              :   REAL;
    xErrorIsOn                  :   BOOL;
    xErrorVerdichterError       :   BOOL;    
    xSafetyStopVerdichter       :   BOOL;    
    TOF_OffToOn                	:   TOF;
	tTimeOffToOn				:	TIME;
    TOF_OnToOn                	:   TOF;
	tTimeOnToOn					: 	TIME;  
    fbVerdichterMotor           :   CtaSysMotor.fbMotor;
    fbCheckVerdichterIsOn       :   CtaSysMotor.fbSafetyInput;    
    fbCheckIsError              :   CtaSysMotor.fbSafetyInput; 
    fbDataCount                 :	CtaSysMotor.fbOperationDataCounter;          
    (* Modbus *)
    xModbusTest                 :   BOOL;
    ayMbControllWord            :   ARRAY[0..3] OF WORD;
    ayMbStateWord               :   ARRAY[0..3] OF WORD;
    (* Einsatzgrenze *)
    ITF_EINSATZGRENZE           :   CtaAppEinsatzDiagramm.ITF_EINSATZGRENZE;
	(* FU *)
	ITF_FU_BASE					:	CtaSysFu.ITF_FU_BASE;
	(* LEISTUNGSVENTILE *)
	ITF_LEISTUNGSVENTILE		:	CtaSysLeistungventile.ITF_LEISTUNGSVENTILE_BASE;
    (* Parameter *)
    fbConfigFile                :   CtaSysConfig.fbConfigFile;
    scParameter                 :   scParameter;
    (* Reports *)	
    fbReportManager			    :   CtaAppReport.fbReportManager;      
    difor					    :	DINT;                                                                    
    ayErrorReporter				:	ARRAY[1..5] OF CtaAppReport.fbReporter;
	ayWarningReporter			:	ARRAY[1..5] OF CtaAppReport.fbReporter;
	(* Trendlog *)
    fbTrendxOn					:	CtaAppInfluxLog.FB_LOG_NODE_BOOL;
	fbTrendxIsOn				:	CtaAppInfluxLog.FB_LOG_NODE_BOOL;
	fbTrendxVerdichterIsOn		:	CtaAppInfluxLog.FB_LOG_NODE_BOOL;
	fbTrendrOnY					:	CtaAppInfluxLog.FB_LOG_NODE_REAL;
	fbTrendrIsOnY				:	CtaAppInfluxLog.FB_LOG_NODE_REAL;
	fbTrendrOnHz				:	CtaAppInfluxLog.FB_LOG_NODE_REAL;
	fbTrendxError				:	CtaAppInfluxLog.FB_LOG_NODE_BOOL;
	(* Collector *)
    diArrayPosition             :   DINT;
END_VAR

(* Config *)
actConfig();

(* Motor Command *)
IF xIsEnabled AND NOT xConfigError THEN
	(* FU *)
	actFU();	
	
    (* Controll Prio *)
    actPrioOfControll();
	
   (* Wiedereinschaltsperre & Pendelschutz*)
    actRestartAndCommutingLock();    
	
    (* Check Compressor is on*)       
    IF scParameter.scInVerdichterOn.fbxDoesAlarm.proValue > scParameter.scInVerdichterOn.fbxEnable.proValue THEN
        // Alarm Only if Enabled
        scParameter.scInVerdichterOn.fbxDoesAlarm.proValue := FALSE;
    END_IF;  
                         
    fbCheckVerdichterIsOn  ((* Inputs *)
                    	xSafetyIn           :=  xVerdichterIsOn,
                    	xReferenceIn        :=  xOn,
                    	(* Parameter *)
                    	fbxEnSafetyInput    :=  scParameter.scInVerdichterOn.fbxDoesAlarm,
                    	fbtStartTime        :=  scParameter.scInVerdichterOn.fbtDelayStart,
                    	fbtRunTime          :=  scParameter.scInVerdichterOn.fbtDelayRun,
                    	(* Outputs *)
                    	xError              =>  xErrorIsOn);  
                    
    (* Check Compressor no error *)
    IF scParameter.scInVerdichterNoError.fbxDoesAlarm.proValue > scParameter.scInVerdichterNoError.fbxEnable.proValue THEN
        // Alarm Only if Enabled
        scParameter.scInVerdichterNoError.fbxDoesAlarm.proValue := FALSE;
    END_IF; 
           
    fbCheckIsError( (* Inputs *)
                    xSafetyIn           :=  xVerdichterNoError,
                    xReferenceIn        :=  TRUE,
                    (* Parameter *)
                    fbxEnSafetyInput    :=  scParameter.scInVerdichterNoError.fbxDoesAlarm,
                    fbtStartTime        :=  scParameter.scInVerdichterNoError.fbtDelayStartSps,
                    fbtRunTime          :=  scParameter.scInVerdichterNoError.fbtDelayRun,
                    (* Outputs *)
                    xError              =>  xErrorVerdichterError);     

    xSafetyStopVerdichter :=  xErrorVerdichterError OR xErrorIsOn OR xSafetyStop;        
    
    (* Scale 0 - 100% *)
	rReleaseScaled  :=	LIMIT(	scParameter.scBase.fbrYMin.rValue,
					    		CtaAppBasic.fcScale(rIn 	:=	CtaAppBasic.fcScale(    rIn                 :=  rVerdichterReleaseY,
																						rMin                :=  0,
																						rMax                :=  100,
																						rOutMin             :=  scHzParameter.rYMinHzAkt,
																						rOutMax             :=  scHzParameter.rYMaxHzAkt),
													rMin	:=	scHzParameter.rYMinHz,
													rMax	:=	scHzParameter.rYMaxHz,
													rOutMin	:=	0,
													rOutMax	:=	100),
								scParameter.scBase.fbrYMax.rValue);
                                                        
    rReleaseScaled  := LIMIT(scParameter.scBase.fbrYMin.proValue , rReleaseScaled ,scParameter.scBase.fbrYMax.proValue); 

    (* Motor *)                
    fbVerdichterMotor  (   (* Inputs *)
                    	xEn                 :=  xVerdiRevisionSwitchOn,
                    	xFreigabe           :=  xReleaseVerdichter,
                    	rFreigabeY          :=  rReleaseScaled,
                    	xSafetyStop         :=  xSafetyStopVerdichter,
                    	(* Parameter *)
                    	fbxEnHandEin        :=  scParameter.scManual.fbxAlowManualOn,
                    	fbxGeregelt         :=  scParameter.scBase.fbxRegulatet,
                    	fbuiHandMode        :=  scParameter.scManual.fbuiManualState,
                    	fbrStellwertHandY   :=  scParameter.scManual.fbrManualOnY,
                    	(* Outputs *)
                    	xOn                 =>  xOn,
                    	rOnY                =>  ,
                    	xHand               =>  );
	
	fbDumperRonY	(	xEn := xOn,
						rSoll := fbVerdichterMotor.rOnY,
						rY => rOnY);	
					
	IF scParameter.scInVerdichterOn.fbxEnable.xValue THEN				
		xIsOn := fbCheckVerdichterIsOn.proOK;
	ELSE
		xIsOn := xOn;
	END_IF
	
	// Check if compressor has valves
	actLeistungsventile();
	
	(*Scale to Hz*)
	rOnHz := 		CtaAppBasic.fcScale	(	rIn 	:= rOnY,
											rMin 	:= 0,
											rMax 	:= 100,
											rOutMin := scHzParameter.rYMinHz,
											rOutMax := scHzParameter.rYMaxHz);
										
	rOnHz := SEL(xOn,0,rOnHz);  

	(*Scale to poweroutput of machine*)
	rOnYVisu :=		LIMIT( 	0,
							CtaAppBasic.fcScale (	rIn 	:= rOnHz,
													rMin 	:= scHzParameter.rYMinHzAkt,
													rMax 	:= scHzParameter.rYMaxHzAkt,
													rOutMin := ((100/SEL(scHzParameter.rYMaxHzAkt = 0,scHzParameter.rYMaxHzAkt,1))*scHzParameter.rYMinHzAkt),
													rOutMax := 100),
							100);
	rOnYVisu := SEL(xOn,0,rOnYVisu);              
        
    (* Data Count Motor *)                                                    
    fbDataCount( xOperating			    := xOn,
                 fbudiOperatingStarts	:= scParameter.scData.fbudiOperationStarts,
                 fbudiOperatingHours	:= scParameter.scData.fbudiOperatingHours);   
                 
    (* EWI *)
    actReport();
	(*Ready output*) 
	xIsReady := xFuseOk AND
				xVerdichterFuseOk AND
				xVerdiRevisionSwitchOn AND
				xVerdichterIsReady AND				
				NOT xOn AND 
				NOT xVerdichterIsOn AND
				NOT xVerdichterHand AND
				NOT TOF_OnToOn.Q AND 
				NOT TOF_OffToOn.Q AND 
				NOT xIsError AND 
				NOT xSafetyStopVerdichter AND
				NOT xIsHandOff AND
				NOT xVerdichterHand AND
				xReadyExt;				             
ELSE
    (* Off if Disabled or Config Error *)
    xOn  		:= FALSE;
    rOnY 		:= 0;
	rOnHz 		:= 0;
	xIsReady := FALSE;    
    (* Reset Flags *)
    actResetOnDisable();
    IF xConfigError THEN
        (* EWI *)
        actReport();         
	END_IF;
END_IF;

(* State *)
actState();

(* Modbus State *)
actMbState();

(* InfluxDB *)
actTrendLog();

ACTION actConfig:
(* Config Fb *)
fbConfigFile();

(* Base Parameter *)
scParameter.scBase.fbxEnable                					(_usiParaNr :=  1, ItfConfigFb := fbConfigFile);
scParameter.scBase.fbxRegulatet             					(_usiParaNr :=  2, ItfConfigFb := fbConfigFile);
scParameter.scBase.fbxEnableFU            						(_usiParaNr :=  3, ItfConfigFb := fbConfigFile);
scParameter.scBase.fbrYMin                  					(_usiParaNr :=  4, ItfConfigFb := fbConfigFile);
scParameter.scBase.fbrYMax                  					(_usiParaNr :=  5, ItfConfigFb := fbConfigFile);
scParameter.scBase.fbtDelayOffToOn              				(_usiParaNr :=  6, ItfConfigFb := fbConfigFile);
scParameter.scBase.fbtDelayOnToOn          						(_usiParaNr :=  7, ItfConfigFb := fbConfigFile);
                                            
(* Fuse Parameter *)                        
scParameter.scFuse.fbxEnable                					(_usiParaNr :=  8, ItfConfigFb := fbconfigFile);
scParameter.scFuse.fbxInputMb               					(_usiParaNr :=  9, ItfConfigFb := fbconfigFile);
scParameter.scFuse.fbxDoesAlarm             					(_usiParaNr := 10, ItfConfigFb := fbconfigFile);
                                            
(* Motor Fuse Parameter *)                  
scParameter.scVerdichterFuse.fbxEnable           				(_usiParaNr := 11, ItfConfigFb := fbconfigFile);
scParameter.scVerdichterFuse.fbxInputMb          				(_usiParaNr := 12, ItfConfigFb := fbconfigFile);
scParameter.scVerdichterFuse.fbxDoesAlarm        				(_usiParaNr := 13, ItfConfigFb := fbconfigFile);
                                            
(* Revision Switch Parameter *)             
scParameter.scInVerdiRevisionSwitch.fbxEnable  					(_usiParaNr := 14, ItfConfigFb := fbconfigFile);
scParameter.scInVerdiRevisionSwitch.fbxInputMb 					(_usiParaNr := 15, ItfConfigFb := fbconfigFile);

(* Motor Input Hand *)
scParameter.scInVerdichterHand.fbxEnable            			(_usiParaNr := 16, ItfConfigFb := fbconfigFile);
scParameter.scInVerdichterHand.fbxInputMb           			(_usiParaNr := 17, ItfConfigFb := fbconfigFile);
                                            
(* Ready Input Parameter *)                 
scParameter.scInVerdichterReady.fbxEnable          		 		(_usiParaNr := 18, ItfConfigFb := fbconfigFile);
scParameter.scInVerdichterReady.fbxInputMb          			(_usiParaNr := 19, ItfConfigFb := fbconfigFile);
                                            
(* Is On Input Parameter *)                 
scParameter.scInVerdichterOn.fbxEnable              			(_usiParaNr := 20, ItfConfigFb := fbconfigFile);
scParameter.scInVerdichterOn.fbxInputMb             			(_usiParaNr := 21, ItfConfigFb := fbconfigFile);
scParameter.scInVerdichterOn.fbxDoesAlarm           			(_usiParaNr := 22, ItfConfigFb := fbconfigFile);
scParameter.scInVerdichterOn.fbtDelayStart          			(_usiParaNr := 23, ItfConfigFb := fbconfigFile);
scParameter.scInVerdichterOn.fbtDelayRun            			(_usiParaNr := 24, ItfConfigFb := fbconfigFile);
scParameter.scInVerdichterOn.fbiTypeOfAck						(_usiParaNr := 25, ItfConfigFb := fbConfigFile,_MinInit := 0,_MaxInit := 2);
scParameter.scInVerdichterOn.fbiMaxErrorRetryAllowed			(_usiParaNr := 26, ItfConfigFb := fbConfigFile); 

(* No Error Input Parameter *)
scParameter.scInVerdichterNoError.fbxEnable         			(_usiParaNr := 27, ItfConfigFb := fbconfigFile);
scParameter.scInVerdichterNoError.fbxInputMb        			(_usiParaNr := 28, ItfConfigFb := fbconfigFile);
scParameter.scInVerdichterNoError.fbxDoesAlarm      			(_usiParaNr := 29, ItfConfigFb := fbconfigFile);
scParameter.scInVerdichterNoError.fbtDelayStartSps  			(_usiParaNr := 30, ItfConfigFb := fbconfigFile);
scParameter.scInVerdichterNoError.fbtDelayRun       			(_usiParaNr := 31, ItfConfigFb := fbconfigFile);
scParameter.scInVerdichterNoError.fbiTypeOfAck					(_usiParaNr := 32, itfConfigFb := fbConfigFile,_MinInit := 0,_MaxInit := 2);
scParameter.scInVerdichterNoError.fbiMaxErrorRetryAllowed		(_usiParaNr := 33, itfConfigFb := fbConfigFile);

(* Actual value Input Parameter *)
scParameter.scInVerdichterActualValue.fbxEnable     			(_usiParaNr := 34, ItfConfigFb := fbconfigFile);
scParameter.scInVerdichterActualValue.fbxInputMb    			(_usiParaNr := 35, ItfConfigFb := fbconfigFile);
scParameter.scInVerdichterActualValue.fbxDoesAlarm  			(_usiParaNr := 36, ItfConfigFb := fbconfigFile);
scParameter.scInVerdichterActualValue.fbrMaxDiff    			(_usiParaNr := 37, ItfConfigFb := fbconfigFile);
scParameter.scInVerdichterActualValue.fbtDelayStart 			(_usiParaNr := 38, ItfConfigFb := fbconfigFile);
scParameter.scInVerdichterActualValue.fbtDelayRun   			(_usiParaNr := 39, ItfConfigFb := fbconfigFile);
scParameter.scInVerdichterActualValue.fbiTypeOfAck				(_usiParaNr := 40, itfConfigFb := fbConfigFile,_MinInit := 0,_MaxInit := 2);
scParameter.scInVerdichterActualValue.fbiMaxErrorRetryAllowed 	(_usiParaNr := 41, itfConfigFb := fbConfigFile);

(* Manual Parameter *)
scParameter.scManual.fbxAlowManualOn        					(_usiParaNr := 42, ItfConfigFb := fbconfigFile); 
scParameter.scManual.fbuiManualState        					(_usiParaNr := 43, ItfConfigFb := fbconfigFile);
scParameter.scManual.fbrManualOnY           					(_usiParaNr := 44, ItfConfigFb := fbconfigFile);

(* Data Counter *)
scParameter.scData.fbudiOperationStarts     					(_usiParaNr := 45, ItfConfigFb := fbconfigFile);
scParameter.scData.fbudiOperatingHours      					(_usiParaNr := 46, ItfConfigFb := fbconfigFile);

(* InfluxDb *)
scParameter.scInfluxDb.fbxEnable            					(_usiParaNr := 47, ItfConfigFb := fbconfigFile);

(* FU *)
scParameter.scFU.fbxReleaseMb									(_usiParaNr := 48, ItfConfigFb := fbconfigFile);
scParameter.scFU.fbxSollWertMb									(_usiParaNr := 49, ItfConfigFb := fbconfigFile);

xConfigError := fbConfigFile.xError;
END_ACTION

PROPERTY proConfigError : BOOL
GET
proConfigError := xConfigError;
END_GET
END_PROPERTY

PROPERTY proAtIconNr : UINT
SET
uiIconNr := proAtIconNr;
END_SET
GET
proAtIconNr:= uiIconNr;
END_GET
END_PROPERTY

PROPERTY P_scBase_fbtDelayOffToOn : CtaSysConfig.ITF_DATATYPE
GET
P_scBase_fbtDelayOffToOn := scParameter.scBase.fbtDelayOffToOn;
END_GET
END_PROPERTY

PROPERTY P_scBase_fbtDelayOnToOn : CtaSysConfig.ITF_DATATYPE
GET
P_scBase_fbtDelayOnToOn := scParameter.scBase.fbtDelayOnToOn;
END_GET
END_PROPERTY

PROPERTY P_scBase_fbrYMax : CtaSysConfig.ITF_DATATYPE
GET
P_scBase_fbrYMax := scParameter.scBase.fbrYMax;
END_GET
END_PROPERTY

PROPERTY P_scBase_fbrYMin : CtaSysConfig.ITF_DATATYPE
GET
P_scBase_fbrYMin := scParameter.scBase.fbrYMin;
END_GET
END_PROPERTY

PROPERTY P_scBase_fbxEnableFU : CtaSysConfig.ITF_DATATYPE
GET
P_scBase_fbxEnableFU := scParameter.scBase.fbxEnableFU;
END_GET
END_PROPERTY

PROPERTY P_scBase_fbxEnable : CtaSysConfig.ITF_DATATYPE
GET
P_scBase_fbxEnable := scParameter.scBase.fbxEnable;
END_GET
END_PROPERTY

PROPERTY P_scBase_fbxRegulatet : CtaSysConfig.ITF_DATATYPE
GET
P_scBase_fbxRegulatet := scParameter.scBase.fbxRegulatet;
END_GET
END_PROPERTY

PROPERTY P_scData_fbudiOperatingHours : CtaSysConfig.ITF_DATATYPE
GET
P_scData_fbudiOperatingHours := scParameter.scData.fbudiOperatingHours;
END_GET
END_PROPERTY

PROPERTY P_scData_fbudiOperationStarts : CtaSysConfig.ITF_DATATYPE
GET
P_scData_fbudiOperationStarts := scParameter.scData.fbudiOperationStarts;
END_GET
END_PROPERTY

PROPERTY P_scFuse_fbxDoesAlarm : CtaSysConfig.ITF_DATATYPE
GET
P_scFuse_fbxDoesAlarm := scParameter.scFuse.fbxDoesAlarm;
END_GET
END_PROPERTY

PROPERTY P_scFuse_fbxEnable : CtaSysConfig.ITF_DATATYPE
GET
P_scFuse_fbxEnable := scParameter.scFuse.fbxEnable;
END_GET
END_PROPERTY

PROPERTY P_scFuse_fbxInputMb : CtaSysConfig.ITF_DATATYPE
GET
P_scFuse_fbxInputMb := scParameter.scFuse.fbxInputMb;
END_GET
END_PROPERTY

PROPERTY P_scInfluxDb_fbxEnable : CtaSysConfig.ITF_DATATYPE
GET
P_scInfluxDb_fbxEnable := scParameter.scInfluxDb.fbxEnable;
END_GET
END_PROPERTY

PROPERTY P_scIO_IsHand_fbxEnable : CtaSysConfig.ITF_DATATYPE
GET
P_scIO_IsHand_fbxEnable := scParameter.scInVerdichterHand.fbxEnable;
END_GET
END_PROPERTY

PROPERTY P_scIO_IsHand_fbxInputMb : CtaSysConfig.ITF_DATATYPE
GET
P_scIO_IsHand_fbxInputMb := scParameter.scInVerdichterHand.fbxInputMb;
END_GET
END_PROPERTY

PROPERTY P_scIO_IsNoError_fbxEnable : CtaSysConfig.ITF_DATATYPE
GET
P_scIO_IsNoError_fbxEnable := scParameter.scInVerdichterNoError.fbxEnable;
END_GET
END_PROPERTY

PROPERTY P_scIO_IsNoError_fbxInputMb : CtaSysConfig.ITF_DATATYPE
GET
P_scIO_IsNoError_fbxInputMb := scParameter.scInVerdichterNoError.fbxInputMb;
END_GET
END_PROPERTY

PROPERTY P_scIO_IsNoError_fbxDoesAlarm : CtaSysConfig.ITF_DATATYPE
GET
P_scIO_IsNoError_fbxDoesAlarm := scParameter.scInVerdichterNoError.fbxDoesAlarm;
END_GET
END_PROPERTY

PROPERTY P_scIO_IsNoError_fbtDelayStartSps : CtaSysConfig.ITF_DATATYPE
GET
P_scIO_IsNoError_fbtDelayStartSps := scParameter.scInVerdichterNoError.fbtDelayStartSps;
END_GET
END_PROPERTY

PROPERTY P_scIO_IsNoError_fbtDelayRun : CtaSysConfig.ITF_DATATYPE
GET
P_scIO_IsNoError_fbtDelayRun := scParameter.scInVerdichterNoError.fbtDelayRun;
END_GET
END_PROPERTY

PROPERTY P_scIO_IsNoError_fbiTypeOfAck : CtaSysConfig.ITF_DATATYPE
GET
P_scIO_IsNoError_fbiTypeOfAck := scParameter.scInVerdichterNoError.fbiTypeOfAck;
END_GET
END_PROPERTY

PROPERTY P_scIO_IsNoError_fbiMaxErrorRetryAllowed : CtaSysConfig.ITF_DATATYPE
GET
P_scIO_IsNoError_fbiMaxErrorRetryAllowed := scParameter.scInVerdichterNoError.fbiMaxErrorRetryAllowed;
END_GET
END_PROPERTY

PROPERTY P_scIO_IsOn_fbxInputMb : CtaSysConfig.ITF_DATATYPE
GET
P_scIO_IsOn_fbxInputMb := scParameter.scInVerdichterOn.fbxInputMb;
END_GET
END_PROPERTY

PROPERTY P_scIO_IsOn_fbxEnable : CtaSysConfig.ITF_DATATYPE
GET
P_scIO_IsOn_fbxEnable := scParameter.scInVerdichterOn.fbxEnable;
END_GET
END_PROPERTY

PROPERTY P_scIO_IsOn_fbtDelayStart : CtaSysConfig.ITF_DATATYPE
GET
P_scIO_IsOn_fbtDelayStart := scParameter.scInVerdichterOn.fbtDelayStart;
END_GET
END_PROPERTY

PROPERTY P_scIO_IsOn_fbxDoesAlarm : CtaSysConfig.ITF_DATATYPE
GET
P_scIO_IsOn_fbxDoesAlarm := scParameter.scInVerdichterOn.fbxDoesAlarm;
END_GET
END_PROPERTY

PROPERTY P_scIO_IsOn_fbtDelayRun : CtaSysConfig.ITF_DATATYPE
GET
P_scIO_IsOn_fbtDelayRun := scParameter.scInVerdichterOn.fbtDelayRun;
END_GET
END_PROPERTY

PROPERTY P_scIO_IsOn_fbiTypeOfAck : CtaSysConfig.ITF_DATATYPE
GET
P_scIO_IsOn_fbiTypeOfAck := scParameter.scInVerdichterOn.fbiTypeOfAck;
END_GET
END_PROPERTY

PROPERTY P_scIO_IsOn_fbiMaxErrorRetryAllowed : CtaSysConfig.ITF_DATATYPE
GET
P_scIO_IsOn_fbiMaxErrorRetryAllowed := scParameter.scInVerdichterOn.fbiMaxErrorRetryAllowed;
END_GET
END_PROPERTY

PROPERTY P_scIO_IsReady_fbxEnable : CtaSysConfig.ITF_DATATYPE
GET
P_scIO_IsReady_fbxEnable := scParameter.scInVerdichterReady.fbxEnable;
END_GET
END_PROPERTY

PROPERTY P_scIO_IsReady_fbxInputMb : CtaSysConfig.ITF_DATATYPE
GET
P_scIO_IsReady_fbxInputMb := scParameter.scInVerdichterReady.fbxInputMb;
END_GET
END_PROPERTY

PROPERTY P_scIO_IsValue_fbxInputMb : CtaSysConfig.ITF_DATATYPE
GET
P_scIO_IsValue_fbxInputMb := scParameter.scInVerdichterActualValue.fbxInputMb;
END_GET
END_PROPERTY

PROPERTY P_scIO_IsValue_fbxEnable : CtaSysConfig.ITF_DATATYPE
GET
P_scIO_IsValue_fbxEnable := scParameter.scInVerdichterActualValue.fbxEnable;
END_GET
END_PROPERTY

PROPERTY P_scIO_IsValue_fbxDoesAlarm : CtaSysConfig.ITF_DATATYPE
GET
P_scIO_IsValue_fbxDoesAlarm := scParameter.scInVerdichterActualValue.fbxDoesAlarm;
END_GET
END_PROPERTY

PROPERTY P_scIO_IsValue_fbtDelayStart : CtaSysConfig.ITF_DATATYPE
GET
P_scIO_IsValue_fbtDelayStart := scParameter.scInVerdichterActualValue.fbtDelayStart;
END_GET
END_PROPERTY

PROPERTY P_scIO_IsValue_fbtDelayRun : CtaSysConfig.ITF_DATATYPE
GET
P_scIO_IsValue_fbtDelayRun := scParameter.scInVerdichterActualValue.fbtDelayRun;
END_GET
END_PROPERTY

PROPERTY P_scIO_IsValue_fbiTypeOfAck : CtaSysConfig.ITF_DATATYPE
GET
P_scIO_IsValue_fbiTypeOfAck := scParameter.scInVerdichterActualValue.fbiTypeOfAck;
END_GET
END_PROPERTY

PROPERTY P_scIO_IsValue_fbiMaxErrorRetryAllowed : CtaSysConfig.ITF_DATATYPE
GET
P_scIO_IsValue_fbiMaxErrorRetryAllowed := scParameter.scInVerdichterActualValue.fbiMaxErrorRetryAllowed;
END_GET
END_PROPERTY

PROPERTY P_scIO_IsValue_fbrMaxDiff : CtaSysConfig.ITF_DATATYPE
GET
P_scIO_IsValue_fbrMaxDiff := scParameter.scInVerdichterActualValue.fbrMaxDiff;
END_GET
END_PROPERTY

PROPERTY P_scIO_RevisionSwitch_fbxEnable : CtaSysConfig.ITF_DATATYPE
GET
P_scIO_RevisionSwitch_fbxEnable := scParameter.scInVerdiRevisionSwitch.fbxEnable;
END_GET
END_PROPERTY

PROPERTY P_scIO_RevisionSwitch_fbxInputMb : CtaSysConfig.ITF_DATATYPE
GET
P_scIO_RevisionSwitch_fbxInputMb := scParameter.scInVerdiRevisionSwitch.fbxInputMb;
END_GET
END_PROPERTY

PROPERTY P_scManual_fbrManualOnY : CtaSysConfig.ITF_DATATYPE
GET
P_scManual_fbrManualOnY := scParameter.scManual.fbrManualOnY;
END_GET
END_PROPERTY

PROPERTY P_scManual_fbuiManualState : CtaSysConfig.ITF_DATATYPE
GET
P_scManual_fbuiManualState := scParameter.scManual.fbuiManualState;
END_GET
END_PROPERTY

PROPERTY P_scManual_fbxAlowManualOn : CtaSysConfig.ITF_DATATYPE
GET
P_scManual_fbxAlowManualOn := scParameter.scManual.fbxAlowManualOn;
END_GET
END_PROPERTY

PROPERTY P_scVerdichterFuse_fbxDoesAlarm : CtaSysConfig.ITF_DATATYPE
GET
P_scVerdichterFuse_fbxDoesAlarm := scParameter.scVerdichterFuse.fbxDoesAlarm;
END_GET
END_PROPERTY

PROPERTY P_scVerdichterFuse_fbxEnable : CtaSysConfig.ITF_DATATYPE
GET
P_scVerdichterFuse_fbxEnable := scParameter.scVerdichterFuse.fbxEnable;
END_GET
END_PROPERTY

PROPERTY P_scVerdichterFuse_fbxInputMb : CtaSysConfig.ITF_DATATYPE
GET
P_scVerdichterFuse_fbxInputMb := scParameter.scVerdichterFuse.fbxInputMb;
END_GET
END_PROPERTY

PROPERTY P_scFU_fbxReleaseMb : CtaSysConfig.ITF_DATATYPE
GET
P_scFU_fbxReleaseMb := scParameter.scFU.fbxReleaseMb;
END_GET
END_PROPERTY

PROPERTY P_scFU_fbxSollWertMb : CtaSysConfig.ITF_DATATYPE
GET
P_scFU_fbxSollWertMb := scParameter.scFU.fbxSollWertMb;
END_GET
END_PROPERTY

PROPERTY proRefToRonYDumper : REFERENCE TO CtaAppDumper.fbDumper
GET
proRefToRonYDumper REF= fbDumperRonY;
END_GET
END_PROPERTY

ACTION actMbState:
IF NOT xModbusTest THEN
    (* State Word 0 Digital Info*)
    ayMbStateWord[0].00     := xOn;
    ayMbStateWord[0].01     := xIsOn;
    ayMbStateWord[0].02     := xVerdichterIsReady;
    ayMbStateWord[0].03     := xVerdichterIsOn;
    ayMbStateWord[0].04     := xVerdichterNoError;
    ayMbStateWord[0].05     := xVerdiRevisionSwitchOn;
    ayMbStateWord[0].06     := xFuseOk;
    ayMbStateWord[0].07     := xVerdichterFuseOk;
    ayMbStateWord[0].08     := xIsHand;
    ayMbStateWord[0].09     := xIsAuto;
    ayMbStateWord[0].10     := FALSE;
    ayMbStateWord[0].11     := FALSE;
    ayMbStateWord[0].12     := FALSE;
    ayMbStateWord[0].13     := FALSE;
    ayMbStateWord[0].14     := xIsWarning;
    ayMbStateWord[0].15     := xIsError;
    (* State Word 1 setpoint*)
    ayMbStateWord[1]        := TO_WORD((TO_INT(rOnYVisu * 10)));
    (* State Word 2 actual value*)
    ayMbStateWord[2]        := SEL(scParameter.scInVerdichterActualValue.fbxEnable.proValue,TO_WORD((TO_INT(rOnYVisu * 10))),
																							TO_WORD((TO_INT(CtaAppBasic.fcScale(rIn 	:= rActualValue,
																																rMin	:= scHzParameter.rYMinHzAkt,
																																rMax 	:= scHzParameter.rYMaxHzAkt,
																																rOutMin := ((scHzParameter.rYMaxHz/100)*scHzParameter.rYMinHz),
																																rOutMax := 100) * 10))));
    (* Hz Aktuell *)
	ayMbStateWord[3]        := SEL(scParameter.scInVerdichterActualValue.fbxEnable.proValue,TO_WORD((TO_INT(rOnHz * 10))),TO_WORD((TO_INT(rActualValue * 10))));

END_IF;
END_ACTION

PROPERTY proModbusTest : BOOL
SET
xModbusTest := proModbusTest;
END_SET
GET
proModbusTest := xModbusTest;
END_GET
END_PROPERTY

{warning disable C0410}
PROPERTY proModbusStateWord : REFERENCE TO ARRAY[0..3] OF WORD
{warning restore C0410}
GET
proModbusStateWord REF= ayMbStateWord;
END_GET
END_PROPERTY

PROPERTY proIsError : BOOL
GET
proIsError := xIsError;
END_GET
END_PROPERTY

PROPERTY proIsWarning : BOOL
GET
proIsWarning := xIsWarning;
END_GET
END_PROPERTY

PROPERTY proIsRegulatet : BOOL
GET
proIsRegulatet := xIsRegulatet;
END_GET
END_PROPERTY

PROPERTY proIsEnabled : BOOL
GET
proIsEnabled := xIsEnabled;
END_GET
END_PROPERTY

ACTION actState:
xIsWarning        := _xIsWarning;         
xIsError          := _xIsError;          
xIsRegulatet      := scParameter.scBase.fbxRegulatet.proValue;         
xIsEnabled        := scParameter.scBase.fbxEnable.proValue;         
xIsHandOn         := scParameter.scManual.fbuiManualState.proValue = 2;         
xIsHandOff        := scParameter.scManual.fbuiManualState.proValue = 1;          
xIsAuto           := scParameter.scManual.fbuiManualState.proValue = 0 AND NOT xVerdichterHand;  
xIsHand           := xIsHandOn OR xIsHandOff OR xVerdichterHand OR xVerdiRevisionSwitchOff;
END_ACTION

PROPERTY proMotorIsOn : BOOL
GET
proMotorIsOn := xVerdichterIsOn OR xIsOn;
END_GET
END_PROPERTY

PROPERTY proIsHandOnOrOff : BOOL
GET
proIsHandOnOrOff := xIsHand;
END_GET
END_PROPERTY

PROPERTY proIsReady : BOOL
GET
proIsReady := xIsReady;
END_GET
END_PROPERTY

PROPERTY proRestartLockAktive : BOOL
GET
proRestartLockAktive := TOF_OffToOn.Q;
END_GET
END_PROPERTY

PROPERTY proCommutingProtectionAktive : BOOL
GET
proCommutingProtectionAktive := TOF_OnToOn.Q;
END_GET
END_PROPERTY

PROPERTY proRevisionSwitchOk : BOOL
GET
proRevisionSwitchOk := xVerdiRevisionSwitchOn;
END_GET
END_PROPERTY

PROPERTY proCountedHours : UDINT
GET
proCountedHours := scParameter.scData.fbudiOperatingHours.proValue;
END_GET
END_PROPERTY

PROPERTY proCountedStarts : UDINT
GET
proCountedStarts := scParameter.scData.fbudiOperationStarts.proValue;
END_GET
END_PROPERTY

PROPERTY proLeistung : REAL
GET
proLeistung := rOnYVisu;
END_GET
END_PROPERTY

PROPERTY proRestartLockTime : TIME
GET
proRestartLockTime := tTimeOffToOn;
END_GET
END_PROPERTY

PROPERTY proCommutingProtectionTime : TIME
GET
proCommutingProtectionTime := tTimeOnToOn;
END_GET
END_PROPERTY

PROPERTY proIsOnY : REAL
GET
proIsOnY := SEL(scParameter.scInVerdichterActualValue.fbxEnable.proValue,rOnY,rInActualValue);
END_GET
END_PROPERTY

PROPERTY proStateSymbol : STRING
GET
IF xIsError THEN
    proStateSymbol := 'CtaVisSymbols.ImagePool.CtaError';
ELSE    
    IF xIsWarning THEN
        IF scEWI.iWarning = 3 THEN
            proStateSymbol := 'CtaVisSymbols.ImagePool.front_hand_Yellow_Off';
        ELSIF scEWI.iWarning = 4 THEN
            proStateSymbol := 'CtaVisSymbols.ImagePool.front_hand_Yellow';
        ELSE
            proStateSymbol := 'CtaVisSymbols.ImagePool.CtaWarning';
        END_IF;
     ELSE
         proStateSymbol := '';
	 END_IF
END_IF;
END_GET
END_PROPERTY

PROPERTY proEnSymbol : STRING
GET
IF xIsEnabled THEN
    proEnSymbol := 'CtaVisSymbols.ImagePool.CheckboxChecked_blue';
ELSE    
    proEnSymbol := 'CtaVisSymbols.ImagePool.CheckboxUnchecked_withe'; 
END_IF;
END_GET
END_PROPERTY

PROPERTY proIsOn : BOOL
GET
proIsOn := xIsOn;
END_GET
END_PROPERTY

PROPERTY proResetVerdiTime : BOOL
SET
IF proResetVerdiTime THEN
	TOF_OnToOn	(PT := T#0S);
	TOF_OffToOn	(PT := T#0S);
END_IF
END_SET
GET
END_GET
END_PROPERTY

PROPERTY proAuto : BOOL
SET
IF proAuto THEN
    scParameter.scManual.fbuiManualState.proValue := 0;
END_IF;
END_SET
GET
proAuto := xIsAuto;
END_GET
END_PROPERTY

PROPERTY proHandOff : BOOL
SET
IF proHandOff THEN
    scParameter.scManual.fbuiManualState.proValue := 1;
END_IF;
END_SET
GET
proHandOff := xIsHandOff;
END_GET
END_PROPERTY

PROPERTY proHandOnY : REAL
GET
proHandOnY := scParameter.scManual.fbrManualOnY.proValue;
END_GET
SET
scParameter.scManual.fbrManualOnY.proValue := proHandOnY;
END_SET
END_PROPERTY

PROPERTY proHardWareHandModulAktive : BOOL
GET
proHardWareHandModulAktive := xVerdichterHand;
END_GET
END_PROPERTY

PROPERTY proHandOn : BOOL
SET
IF proHandOn THEN
    scParameter.scManual.fbuiManualState.proValue := 2;
END_IF;
END_SET
GET
proHandOn := xIsHandOn;
END_GET
END_PROPERTY

PROPERTY proGetDI_IsOn : BOOL
GET
proGetDI_IsOn := xInVerdichterIsOn;
END_GET
END_PROPERTY

METHOD metDI_IsOn
VAR_INPUT
	ITF_IN		:	CtaSysIO.ITF_IO;	    
END_VAR
VAR	
	ITF_DI		:	CtaSysIO.ITF_DI;
END_VAR
IF ITF_IN <> 0 THEN
	ITF_VerdichterIsOn := ITF_IN;	
	IF __QUERYINTERFACE(ITF_VerdichterIsOn,ITF_DI) THEN		
		xInVerdichterIsOn := ITF_DI.proValue;
	END_IF	
ELSE
	xinVerdichterIsOn := FALSE;
END_IF
END_METHOD

PROPERTY proNotShowDI_IsOn : BOOL
GET
proNotShowDI_IsOn := NOT scParameter.scInVerdichterOn.fbxEnable.xValue OR scParameter.scInVerdichterOn.fbxInputMb.xValue;
END_GET
END_PROPERTY

PROPERTY proIsOn_ITF : CtaSysIO.ITF_IO
GET
proIsOn_ITF := ITF_VerdichterIsOn;
END_GET
END_PROPERTY

METHOD metDI_RevisionSwitchOk
VAR_INPUT
    ITF_IN		:	CtaSysIO.ITF_IO;
END_VAR
VAR	
	ITF_DI		:	CtaSysIO.ITF_DI;
END_VAR
IF ITF_IN <> 0 THEN	
	ITF_RevisionSwitch := ITF_IN;
	IF __QUERYINTERFACE(ITF_RevisionSwitch,ITF_DI) THEN		
		xInVerdiRevisionSwitchOn := ITF_DI.proValue;
	END_IF	
ELSE
	xInVerdiRevisionSwitchOn := FALSE;
END_IF
END_METHOD

PROPERTY proNotShowDI_RevisionSwitchOk : BOOL
GET
proNotShowDI_RevisionSwitchOk := NOT scParameter.scInVerdiRevisionSwitch.fbxEnable.xValue OR scParameter.scInVerdiRevisionSwitch.fbxInputMb.xValue;
END_GET
END_PROPERTY

PROPERTY proGetDI_RevisionSwitchOK : BOOL
GET
proGetDI_RevisionSwitchOK := xInVerdiRevisionSwitchOn;
END_GET
END_PROPERTY

PROPERTY proRevisionSwitch_ITF : CtaSysIO.ITF_IO
GET
proRevisionSwitch_ITF := ITF_RevisionSwitch;
END_GET
END_PROPERTY

METHOD metDI_NoError
VAR_INPUT
    ITF_IN		:	CtaSysIO.ITF_IO;
END_VAR
VAR	
	ITF_DI		:	CtaSysIO.ITF_DI;
END_VAR
IF ITF_IN <> 0 THEN
	ITF_VerdichterNoError := ITF_IN;	
	IF __QUERYINTERFACE(ITF_VerdichterNoError,ITF_DI) THEN		
		xInVerdichterNoError := ITF_DI.proValue;
	END_IF	
ELSE
	xInVerdichterNoError := FALSE;
END_IF
END_METHOD

PROPERTY proNotShowDI_NoError : BOOL
GET
proNotShowDI_NoError := NOT scParameter.scInVerdichterNoError.fbxEnable.xValue OR scParameter.scInVerdichterNoError.fbxInputMb.xValue;
END_GET
END_PROPERTY

PROPERTY proGetDI_NoError : BOOL
GET
proGetDI_NoError := xInVerdichterNoError;
END_GET
END_PROPERTY

PROPERTY proNoError_ITF : CtaSysIO.ITF_IO
GET
proNoError_ITF := ITF_VerdichterNoError;
END_GET
END_PROPERTY

PROPERTY proGetDI_FuseOK : BOOL
GET
proGetDI_FuseOK := xInFuseOk;
END_GET
END_PROPERTY

METHOD metDI_ITF_FuseOK
VAR_INPUT
	ITF_IN		:	CtaSysIO.ITF_IO;	
END_VAR
VAR
	ITF_DI		:	CtaSysIO.ITF_DI;
END_VAR
IF ITF_IN <> 0 THEN
	ITF_Fuse := ITF_IN; 
	IF __QUERYINTERFACE(ITF_Fuse,ITF_DI) THEN		
		xInFuseOk := ITF_DI.proValue;
	END_IF	
ELSE
	xInFuseOk := FALSE;
END_IF
END_METHOD

PROPERTY proNotShowDI_FuseOk : BOOL
GET
proNotShowDI_FuseOk := NOT scParameter.scFuse.fbxEnable.xValue OR scParameter.scFuse.fbxInputMb.xValue;
END_GET
END_PROPERTY

PROPERTY proFuse_ITF : CtaSysIO.ITF_IO
GET
proFuse_ITF := ITF_Fuse;
END_GET
END_PROPERTY

METHOD metDI_ITF_VerdichterHand
VAR_INPUT
	ITF_IN		:	CtaSysIO.ITF_IO;	
END_VAR
VAR	
	ITF_DI		:	CtaSysIO.ITF_DI;
END_VAR
IF ITF_IN <> 0 THEN	
	ITF_VerdichterHand := ITF_IN;
	IF __QUERYINTERFACE(ITF_VerdichterHand,ITF_DI) THEN		
		xinVerdichterHand := ITF_DI.proValue;
	END_IF	
ELSE
	xInVerdichterHand := FALSE;
END_IF
END_METHOD

PROPERTY proNotShowDI_VerdichterHand : BOOL
GET
proNotShowDI_VerdichterHand := NOT scParameter.scInVerdichterHand.fbxEnable.xValue OR scParameter.scInVerdichterHand.fbxInputMb.xValue;
END_GET
END_PROPERTY

PROPERTY proGetDI_VerdichterHand : BOOL
GET
proGetDI_VerdichterHand := xInVerdichterHand;
END_GET
END_PROPERTY

PROPERTY proHandModul_ITF : CtaSysIO.ITF_IO
GET
proHandModul_ITF := ITF_VerdichterHand;
END_GET
END_PROPERTY

METHOD metDI_IsReady
VAR_INPUT
    ITF_IN		:	CtaSysIO.ITF_IO;
END_VAR
VAR	
	ITF_DI		:	CtaSysIO.ITF_DI;
END_VAR
IF ITF_IN <> 0 THEN	
	ITF_VerdichterIsReady := ITF_IN;
	IF __QUERYINTERFACE(ITF_VerdichterIsReady,ITF_DI) THEN		
		xInVerdichterIsReady := ITF_DI.proValue;
	END_IF	
ELSE
	xInVerdichterIsReady := FALSE;
END_IF
END_METHOD

PROPERTY proNotShowDI_Ready : BOOL
GET
proNotShowDI_Ready := NOT scParameter.scInVerdichterReady.fbxEnable.xValue OR scParameter.scInVerdichterReady.fbxInputMb.xValue;
END_GET
END_PROPERTY

PROPERTY proGetDI_IsReady : BOOL
GET
proGetDI_IsReady := xInVerdichterIsReady;
END_GET
END_PROPERTY

PROPERTY proReady_ITF : CtaSysIO.ITF_IO
GET
proReady_ITF := ITF_VerdichterIsReady;
END_GET
END_PROPERTY

METHOD metDI_VerdichterFuseOk
VAR_INPUT
    ITF_IN		:	CtaSysIO.ITF_IO;
END_VAR
VAR	
	ITF_DI		:	CtaSysIO.ITF_DI;
END_VAR
IF ITF_IN <> 0 THEN
	ITF_VerdichterFuse := ITF_IN;	
	IF __QUERYINTERFACE(ITF_VerdichterFuse,ITF_DI) THEN		
		xInVerdichterFuseOk := ITF_DI.proValue;
	END_IF	
ELSE
	xInVerdichterFuseOk := FALSE;
END_IF
END_METHOD

PROPERTY proNotShowDI_VerdichterFuseOk : BOOL
GET
proNotShowDI_VerdichterFuseOk := NOT scParameter.scVerdichterFuse.fbxEnable.xValue OR scParameter.scVerdichterFuse.fbxInputMb.xValue;
END_GET
END_PROPERTY

PROPERTY proGetDI_VerdichterFuseOk : BOOL
GET
proGetDI_VerdichterFuseOk := xInVerdichterFuseOk;
END_GET
END_PROPERTY

PROPERTY proVerdichterFuse_ITF : CtaSysIO.ITF_IO
GET
proVerdichterFuse_ITF := ITF_VerdichterFuse;
END_GET
END_PROPERTY

METHOD metAI_ActualValue
VAR_INPUT
    ITF_IN		:	CtaSysIO.ITF_IO;
END_VAR
VAR	
	ITF_AI		:	CtaSysIO.ITF_AI;
END_VAR
IF ITF_IN <> 0 THEN
	ITF_ActualValue := ITF_IN;	
	IF __QUERYINTERFACE(ITF_ActualValue,ITF_AI) THEN		
		rInActualValue := ITF_AI.proValue;
	END_IF	
ELSE
	rInActualValue := 0;
END_IF
END_METHOD

PROPERTY proGetAI_ActualValue : REAL
GET
proGetAI_ActualValue := rInActualValue;
END_GET
END_PROPERTY

PROPERTY proNotShowAI_ActualValue : BOOL
GET
proNotShowAI_ActualValue := NOT scParameter.scInVerdichterActualValue.fbxEnable.xValue OR scParameter.scFuse.fbxInputMb.xValue;
END_GET
END_PROPERTY

PROPERTY proActualValue_ITF : CtaSysIO.ITF_IO
GET
proActualValue_ITF := ITF_ActualValue;
END_GET
END_PROPERTY

PROPERTY proOnY_ITF : CtaSysIO.ITF_IO
GET
proOnY_ITF := ITF_rOnY;
END_GET
END_PROPERTY

METHOD metAO_OnY : REAL
VAR_INPUT
    ITF_IN		:	CtaSysIO.ITF_IO;
END_VAR
VAR	
	ITF_AO		:	CtaSysIO.ITF_AO;
END_VAR
IF ITF_IN <> 0 THEN
	ITF_rOnY := ITF_IN;	
	IF __QUERYINTERFACE(ITF_rOnY,ITF_AO) THEN		
		ITF_AO.proValue := rOnY;
	END_IF	
ELSE
	metAO_OnY := rOnY;
END_IF
END_METHOD

PROPERTY proDO_On : BOOL
GET
proDO_On := xOn;
END_GET
END_PROPERTY

METHOD metDO_On : BOOL
VAR_INPUT
    ITF_IN		:	CtaSysIO.ITF_IO;
END_VAR
VAR	
	ITF_DO		:	CtaSysIO.ITF_DO;
END_VAR
IF ITF_IN <> 0 THEN	
	ITF_xOn := ITF_IN;
	IF __QUERYINTERFACE(ITF_xOn,ITF_DO) THEN		
		ITF_DO.proValue := xOn;
	END_IF	
ELSE
	metDO_On := xOn;
END_IF
END_METHOD

PROPERTY proOn_ITF : CtaSysIO.ITF_IO
GET
proOn_ITF := ITF_xOn;
END_GET
END_PROPERTY

PROPERTY proOnY : REAL
GET
proOnY := rOnY;
END_GET
END_PROPERTY

PROPERTY proOn : BOOL
GET
proOn := xOn;
END_GET
END_PROPERTY

ACTION actRestartAndCommutingLock:
(*Wiedereinschaltsperre*)
TOF_OffToOn	(	PT  :=  scParameter.scBase.fbtDelayOffToOn.proValue,
				IN  := NOT xOn AND xOnOld);
tTimeOffToOn := scParameter.scBase.fbtDelayOffToOn.proValue - TOF_OffToOn.ET; 
         
(*Pendelschutz*)
TOF_OnToOn	(   PT  :=  scParameter.scBase.fbtDelayOnToOn.proValue,
				IN  :=  xOn AND NOT xOnOld);     
tTimeOnToOn := scParameter.scBase.fbtDelayOnToOn.proValue - TOF_OnToOn.ET;

(*Alten Wert zwischenspeichern*)
xOnOld := xOn;
END_ACTION

ACTION actPrioOfControll:
(*Release for Compressor only from physical inputs*)
xReleaseVerdichter 	:= xRelease AND (xOn OR (NOT TOF_OffToOn.Q AND NOT TOF_OnToOn.Q)) AND NOT xIsError;	
rVerdichterReleaseY := rRelease;

(* Get state from Input or ModBus *)
(* Fuse ok *)
// Flag FuseOk True if not Enabled
xFuseOk                            		:= SEL(scParameter.scFuse.fbxEnable.xValue                   ,TRUE   ,SEL(scParameter.scFuse.fbxInputMb.xValue               		,xInFuseOk                  ,xInFuseOkMb                	));                     
(* Motor fuse ok *)
// Flag MotorFuseOk True if not Enabled
xVerdichterFuseOk                       := SEL(scParameter.scVerdichterFuse.fbxEnable.xValue         ,TRUE   ,SEL(scParameter.scVerdichterFuse.fbxInputMb.xValue          	,xInVerdichterFuseOk        ,xInVerdichterFuseOkMb          ));
(* Motor is hand *)
// Flag MotorHand False if not Enabled
xVerdichterHand                         := SEL(scParameter.scInVerdichterHand.fbxEnable.xValue       ,FALSE  ,SEL(scParameter.scInVerdichterHand.fbxInputMb.xValue          ,xInVerdichterHand          ,xInVerdichterHandMb            ));  
(* Motor is ready *)
// Flag MotorIsReady True if not Enabled
xVerdichterIsReady                      := SEL(scParameter.scInVerdichterReady.fbxEnable.xValue      ,TRUE   ,SEL(scParameter.scInVerdichterReady.fbxInputMb.xValue         ,xInVerdichterIsReady       ,xInVerdichterIsReadyMb         )); 
(* Motor is on *)
// Flag MotorIsOn False if not Enabled
xVerdichterIsOn                         := SEL(scParameter.scInVerdichterOn.fbxEnable.xValue         ,FALSE  ,SEL(scParameter.scInVerdichterOn.fbxInputMb.xValue        	,xInVerdichterIsOn          ,xInVerdichterIsOnMb            ));  
(* Motor no error *)
// Flag MotorNoError True if not Enabled
xVerdichterNoError                      := SEL(scParameter.scInVerdichterNoError.fbxEnable.xValue    ,TRUE   ,SEL(scParameter.scInVerdichterNoError.fbxInputMb.xValue       ,xInVerdichterNoError       ,xInVerdichterNoErrorMb        	));
(* Revision Switch *)
// Flag MotorRevisionSwitchOn True if not Enabled
xVerdiRevisionSwitchOn             		:= SEL(scParameter.scInVerdiRevisionSwitch.fbxEnable.xValue  ,TRUE   ,SEL(scParameter.scInVerdiRevisionSwitch.fbxInputMb.xValue		,xInVerdiRevisionSwitchOn	,xInVerdiRevisionSwitchOnMb 	));
xVerdiRevisionSwitchOff            		:= NOT xVerdiRevisionSwitchOn;
END_ACTION

ACTION actResetOnDisable:
(* Reset Lead and Run After Command *)
    TOF_OffToOn.PT           := T#0MS;
    TOF_OffToOn.IN           := FALSE;  
    TOF_OffToOn();           
    TOF_OnToOn.PT            := T#0MS;
    TOF_OnToOn.IN            := FALSE;  
    TOF_OnToOn();               
    xReleaseVerdichter       := FALSE;
    xIsOn                    := FALSE;
    xFuseOk                  := FALSE;    
    xVerdichterFuseOk        := FALSE;
    xVerdichterNoError       := FALSE;
    xVerdichterIsReady       := FALSE;
    xVerdiRevisionSwitchOn   := FALSE;
    xVerdichterIsOn          := FALSE;
    xVerdichterHand          := FALSE;
	rActualValue			 := 	0;
END_ACTION

PROPERTY proOnHz : REAL
GET
proOnHz := rOnHz;
END_GET
END_PROPERTY

PROPERTY proEn : BOOL
SET
xIsEnabled := proEn;
END_SET
GET
proEn := xIsEnabled;
END_GET
END_PROPERTY

ACTION actTrendLog:
(* Schaltbefehl *)
fbTrendxOn.ENABLE					:=	scParameter.scBase.fbxEnable.proValue AND
										scParameter.scInfluxDb.fbxEnable.proValue;
fbTrendxOn.KEY						:=	CONCAT(stObjID,'_xOn');
fbTrendxOn.SET_VALUE				:=  xOn;

(* Betriebsmeldung *)
fbTrendxIsOn.ENABLE					:=	scParameter.scBase.fbxEnable.proValue AND
										scParameter.scInfluxDb.fbxEnable.proValue;
fbTrendxIsOn.KEY					:=	CONCAT(stObjID,'_xIsOn');
fbTrendxIsOn.SET_VALUE				:=	xIsOn;

(* Betriebsmeldung Motor *)
fbTrendxVerdichterIsOn.ENABLE		:=	scParameter.scBase.fbxEnable.proValue AND
										scParameter.scInfluxDb.fbxEnable.proValue;
fbTrendxVerdichterIsOn.KEY			:=	CONCAT(stObjID,'_xVerdichterIsOn');
fbTrendxVerdichterIsOn.SET_VALUE	:=	xVerdichterIsOn;

(* Stellwert *)
fbTrendrOnY.ENABLE					:=	scParameter.scBase.fbxEnable.proValue AND
										scParameter.scInfluxDb.fbxEnable.proValue;
fbTrendrOnY.KEY						:=	CONCAT(stObjID,'_rOnY');
fbTrendrOnY.SET_VALUE				:= 	rOnY; 

(* Istwert *)
fbTrendrIsOnY.ENABLE				:=	scParameter.scBase.fbxEnable.proValue AND
										scParameter.scInfluxDb.fbxEnable.proValue;
fbTrendrIsOnY.KEY					:=	CONCAT(stObjID,'_rIsOnY');
fbTrendrIsOnY.SET_VALUE				:= 	proIsOnY;

(* Hz *)
fbTrendrOnHz.ENABLE					:=	scParameter.scBase.fbxEnable.proValue AND
										scParameter.scInfluxDb.fbxEnable.proValue;
fbTrendrOnHz.KEY					:=	CONCAT(stObjID,'_rOnHz');
fbTrendrOnHz.SET_VALUE				:=  proOnHz;

(* Fehler *)
fbTrendxError.ENABLE				:=	scParameter.scBase.fbxEnable.proValue AND
										scParameter.scInfluxDb.fbxEnable.proValue;
fbTrendxError.KEY					:=	CONCAT(stObjID,'_xError');
fbTrendxError.SET_VALUE				:=  xIsError;
END_ACTION

ACTION actReport:
(* EWI Manager *)
fbReportManager(	stErrorInitReportTextListIn		:=	ADR(GlobalKonstant.stReportTextListError),
					stWarningInitReportTextListIn	:=	ADR(GlobalKonstant.stReportTextListWarning),
					stInfoInitReportTextListIn		:=	ADR(GlobalKonstant.stReportTextListInfo),
					scReportNr						:=	scEWI);
(* Errors *)                        
        (* Meldung Error On *)
        ayErrorReporter[1].proPrio  := 3;
        ayErrorReporter[1].metReport(     		xSetReportIn					:= xErrorIsOn AND scParameter.scInVerdichterOn.fbxDoesAlarm.proValue AND scParameter.scInVerdichterOn.fbxEnable.proValue,
												iReportID						:= 1,
												enReportTypeIn					:= CtaAppReport.enReportType.Error,  
												enReportAcknowledgeTypeIn   	:= scParameter.scInVerdichterOn.fbiTypeOfAck.proValue,
												tDelay							:= T#0S, 
												ITF_BMK_IN						:= THIS^,			              
												pstReportTextListIn				:= ADR(GlobalKonstant.stReportTextListError),
												stOptionalReportText		    := '',   
												iRetryTilReportLock 		    := scParameter.scInVerdichterOn.fbiMaxErrorRetryAllowed.proValue, 
												xResetCount         		    := FALSE,  
												tReset						    := T#24H); 		

        (* Error Motor *)    
        ayErrorReporter[2].proPrio  := 3;
        ayErrorReporter[2].metReport(     		xSetReportIn					:= xErrorVerdichterError AND scParameter.scInVerdichterNoError.fbxDoesAlarm.proValue AND scParameter.scInVerdichterNoError.fbxEnable.proValue,
												iReportID						:= 2,
												enReportTypeIn					:= CtaAppReport.enReportType.Error,  
												enReportAcknowledgeTypeIn   	:= scParameter.scInVerdichterNoError.fbiTypeOfAck.proValue,
												tDelay							:= T#0S, 
												ITF_BMK_IN						:= THIS^,			              
												pstReportTextListIn				:= ADR(GlobalKonstant.stReportTextListError),
												stOptionalReportText		    := '',   
												iRetryTilReportLock 		    := scParameter.scInVerdichterNoError.fbiMaxErrorRetryAllowed.proValue, 
												xResetCount         		    := FALSE,  
												tReset						    := T#24H); 	  
                           
        (* Error Fuse *) 
        ayErrorReporter[3].proPrio  := 2;   
        ayErrorReporter[3].metReport(     		xSetReportIn					:= NOT xFuseOk AND scParameter.scFuse.fbxDoesAlarm.proValue AND scParameter.scFuse.fbxEnable.proValue,
												iReportID						:= 3,
												enReportTypeIn					:= CtaAppReport.enReportType.Error,  
												enReportAcknowledgeTypeIn   	:= CtaAppReport.enReportacknowledgeType.Auto,
												tDelay							:= T#1S, 
												ITF_BMK_IN						:= THIS^,			              
												pstReportTextListIn				:= ADR(GlobalKonstant.stReportTextListError),
												stOptionalReportText		    := '',   
												iRetryTilReportLock 		    := 0, 
												xResetCount         		    := FALSE,  
												tReset						    := T#24H);
                                                
        (* Error Motor Fuse *)    
        ayErrorReporter[4].proPrio  := 2;
        ayErrorReporter[4].metReport(     		xSetReportIn					:= NOT xVerdichterFuseOk AND scParameter.scVerdichterFuse.fbxDoesAlarm.proValue AND scParameter.scVerdichterFuse.fbxEnable.proValue,
												iReportID						:= 4,
												enReportTypeIn					:= CtaAppReport.enReportType.Error,  
												enReportAcknowledgeTypeIn   	:= CtaAppReport.enReportacknowledgeType.Auto,
												tDelay							:= T#1S, 
												ITF_BMK_IN						:= THIS^,			              
												pstReportTextListIn				:= ADR(GlobalKonstant.stReportTextListError),
												stOptionalReportText		    := '',   
												iRetryTilReportLock 		    := 0, 
												xResetCount         		    := FALSE,  
												tReset						    := T#24H);                                                

        (* Config Error *)    
        ayErrorReporter[5].proPrio  := 1;
        ayErrorReporter[5].metReport(     		xSetReportIn					:= xConfigError,
												iReportID						:= 5,
												enReportTypeIn					:= CtaAppReport.enReportType.Error,  
												enReportAcknowledgeTypeIn   	:= CtaAppReport.enReportacknowledgeType.Quit,
												tDelay							:= T#1S, 
												ITF_BMK_IN						:= THIS^,			              
												pstReportTextListIn				:= ADR(GlobalKonstant.stReportTextListError),
												stOptionalReportText		    := '',   
												iRetryTilReportLock 		    := 0, 
												xResetCount         		    := FALSE,  
												tReset						    := T#24H);                                           
(* Warnungen *)      
        (* Warnung Sicherheits Stopp *)      
        ayWarningReporter[1].proPrio := 2;
        ayWarningReporter[1].metReport(			xSetReportIn					:= xSafetyStopVerdichter AND xReleaseVerdichter,
												iReportID						:= 1,
												enReportTypeIn					:= CtaAppReport.enReportType.Warning,  
												enReportAcknowledgeTypeIn   	:= CtaAppReport.enReportAcknowledgeType.Auto,
												tDelay							:= T#0S, 
												ITF_BMK_IN						:= THIS^,			              
												pstReportTextListIn				:= ADR(GlobalKonstant.stReportTextListWarning),
												stOptionalReportText		    := '',   
												iRetryTilReportLock 		    := 0, 
												xResetCount         		    := FALSE,  
												tReset						    := T#24H);                       
                                  
